LIN {X 0,Y 580.036,Z 777.996,A -85,B 0,C 180,E1 -1980,E2 -1980} C_VEL
LIN {X 0,Y 580.038,Z 777.751,A -85,B 0,C 180,E1 -1980.694,E2 -1980.694} C_VEL
LIN {X 0,Y 580.046,Z 776.958,A -85,B 0,C 180,E1 -1981.389,E2 -1981.389} C_VEL
LIN {X 0,Y 580.034,Z 775.61,A -85,B 0,C 180,E1 -1982.083,E2 -1982.083} C_VEL
LIN {X 0,Y 580.073,Z 772.575,A -85,B 0,C 180,E1 -1983.125,E2 -1983.125} C_VEL
LIN {X 0,Y 580.109,Z 768.035,A -85,B 0,C 180,E1 -1984.169,E2 -1984.169} C_VEL
LIN {X 0,Y 580.127,Z 762.947,A -85,B 0,C 180,E1 -1985.039,E2 -1985.039} C_VEL
LIN {X 0,Y 580.195,Z 756.461,A -85,B 0,C 180,E1 -1985.91,E2 -1985.91} C_VEL
LIN {X 0,Y 580.226,Z 747.843,A -85,B 0,C 180,E1 -1986.806,E2 -1986.806} C_VEL
LIN {X 0,Y 580.271,Z 739.422,A -85,B 0,C 180,E1 -1987.481,E2 -1987.481} C_VEL
LIN {X 0,Y 580.361,Z 729.698,A -85,B 0,C 180,E1 -1988.093,E2 -1988.093} C_VEL
LIN {X 0,Y 580.434,Z 719.272,A -85,B 0,C 180,E1 -1988.574,E2 -1988.574} C_VEL
LIN {X 0,Y 580.421,Z 709.143,A -85,B 0,C 180,E1 -1988.903,E2 -1988.903} C_VEL
LIN {X 0,Y 580.451,Z 698.454,A -85,B 0,C 180,E1 -1989.122,E2 -1989.122} C_VEL
LIN {X 0,Y 580.405,Z 632.513,A -85,B 0,C 180,E1 -1989.936,E2 -1989.936} C_VEL
LIN {X 0,Y 580.269,Z 630.726,A -85,B 0,C 180,E1 -1990.005,E2 -1990.005} C_VEL
LIN {X 0,Y 580.35,Z 617.125,A -85,B 0,C 180,E1 -1991.689,E2 -1991.689} C_VEL
LIN {X 0,Y 579.697,Z 613.548,A -85,B 0,C 180,E1 -1992.149,E2 -1992.149} C_VEL
LIN {X 0,Y 574.108,Z 602.38,A -85,B 0,C 180,E1 -1993.683,E2 -1993.683} C_VEL
LIN {X 0,Y 573.454,Z 598.82,A -85,B 0,C 180,E1 -1994.152,E2 -1994.152} C_VEL
LIN {X 0,Y 573.677,Z 575.438,A -85,B 0,C 180,E1 -1997.144,E2 -1997.144} C_VEL
LIN {X 0,Y 573.912,Z 553.049,A -85,B 0,C 180,E1 -2000.053,E2 -2000.053} C_VEL
LIN {X 0,Y 574.175,Z 533.149,A -85,B 0,C 180,E1 -2002.679,E2 -2002.679} C_VEL
LIN {X 0,Y 574.39,Z 518.935,A -85,B 0,C 180,E1 -2004.583,E2 -2004.583} C_VEL
LIN {X 0,Y 573.29,Z 513.146,A -85,B 0,C 180,E1 -2005.457,E2 -2005.457} C_VEL
LIN {X 0,Y 573.252,Z 513.079,A -85,B 0,C 180,E1 -2008.028,E2 -2008.028} C_VEL
LIN {X 0,Y 573.25,Z 513.08,A -85,B 0,C 180,E1 -2010.176,E2 -2010.176} C_VEL
LIN {X 0,Y 573.258,Z 513.079,A -85,B 0,C 180,E1 -2012.645,E2 -2012.645} C_VEL
LIN {X 0,Y 573.272,Z 513.071,A -85,B 0,C 180,E1 -2015.184,E2 -2015.184} C_VEL
LIN {X 0,Y 573.24,Z 513.075,A -85,B 0,C 180,E1 -2017.807,E2 -2017.807} C_VEL
LIN {X 0,Y 573.275,Z 513.076,A -85,B 0,C 180,E1 -2020.528,E2 -2020.528} C_VEL
LIN {X 0,Y 573.248,Z 513.069,A -85,B 0,C 180,E1 -2023.669,E2 -2023.669} C_VEL
LIN {X 0,Y 573.252,Z 513.081,A -85,B 0,C 180,E1 -2026.642,E2 -2026.642} C_VEL
LIN {X 0,Y 573.249,Z 513.07,A -85,B 0,C 180,E1 -2029.475,E2 -2029.475} C_VEL
LIN {X 0,Y 573.241,Z 513.076,A -85,B 0,C 180,E1 -2032.192,E2 -2032.192} C_VEL
LIN {X 0,Y 573.239,Z 513.074,A -85,B 0,C 180,E1 -2035.229,E2 -2035.229} C_VEL
LIN {X 0,Y 573.257,Z 513.072,A -85,B 0,C 180,E1 -2037.771,E2 -2037.771} C_VEL
LIN {X 0,Y 573.269,Z 513.081,A -85,B 0,C 180,E1 -2040.634,E2 -2040.634} C_VEL
LIN {X 0,Y 573.256,Z 513.077,A -85,B 0,C 180,E1 -2043.024,E2 -2043.024} C_VEL
LIN {X 0,Y 573.281,Z 513.068,A -85,B 0,C 180,E1 -2045.366,E2 -2045.366} C_VEL
LIN {X 0,Y 573.234,Z 513.081,A -85,B 0,C 180,E1 -2048.419,E2 -2048.419} C_VEL
LIN {X 0,Y 573.317,Z 513.261,A -85,B 0,C 180,E1 -2050.276,E2 -2050.276} C_VEL
LIN {X 0,Y 573.558,Z 518.552,A -85,B 0,C 180,E1 -2051.237,E2 -2051.237} C_VEL
LIN {X 0,Y 573.387,Z 536.372,A -85,B 0,C 180,E1 -2054.356,E2 -2054.356} C_VEL
LIN {X 0,Y 573.308,Z 547.196,A -85,B 0,C 180,E1 -2056.192,E2 -2056.192} C_VEL
LIN {X 0,Y 573.776,Z 550.135,A -85,B 0,C 180,E1 -2056.277,E2 -2056.277} C_VEL
LIN {X 0,Y 574.078,Z 556.84,A -85,B 0,C 180,E1 -2056.369,E2 -2056.369} C_VEL
LIN {X 0,Y 573.884,Z 653.913,A -85,B 0,C 180,E1 -2057.602,E2 -2057.602} C_VEL
LIN {X 0,Y 573.815,Z 667.2,A -85,B 0,C 180,E1 -2057.915,E2 -2057.915} C_VEL
LIN {X 0,Y 573.718,Z 679.359,A -85,B 0,C 180,E1 -2058.339,E2 -2058.339} C_VEL
LIN {X 0,Y 573.588,Z 690.955,A -85,B 0,C 180,E1 -2058.881,E2 -2058.881} C_VEL
LIN {X 0,Y 573.447,Z 702.545,A -85,B 0,C 180,E1 -2059.585,E2 -2059.585} C_VEL
LIN {X 0,Y 573.332,Z 713.057,A -85,B 0,C 180,E1 -2060.385,E2 -2060.385} C_VEL
LIN {X 0,Y 573.242,Z 721.659,A -85,B 0,C 180,E1 -2061.184,E2 -2061.184} C_VEL
LIN {X 0,Y 573.162,Z 729.582,A -85,B 0,C 180,E1 -2062.07,E2 -2062.07} C_VEL
LIN {X 0,Y 573.092,Z 737.519,A -85,B 0,C 180,E1 -2063.162,E2 -2063.162} C_VEL
LIN {X 0,Y 573.071,Z 744.446,A -85,B 0,C 180,E1 -2064.369,E2 -2064.369} C_VEL
LIN {X 0,Y 573.028,Z 749.188,A -85,B 0,C 180,E1 -2065.427,E2 -2065.427} C_VEL
LIN {X 0,Y 573.022,Z 752.821,A -85,B 0,C 180,E1 -2066.484,E2 -2066.484} C_VEL
LIN {X 0,Y 572.959,Z 754.699,A -85,B 0,C 180,E1 -2067.187,E2 -2067.187} C_VEL
LIN {X 0,Y 572.939,Z 756.128,A -85,B 0,C 180,E1 -2067.89,E2 -2067.89} C_VEL
LIN {X 0,Y 572.941,Z 757.755,A -85,B 0,C 180,E1 -2069.297,E2 -2069.297} C_VEL
LIN {X 0,Y 572.939,Z 757.996,A -85,B 0,C 180,E1 -2069.999,E2 -2069.999} C_VEL
LIN {X 0,Y 572.94,Z 757.815,A -85,B 0,C 180,E1 -2070.702,E2 -2070.702} C_VEL
LIN {X 0,Y 572.939,Z 756.273,A -85,B 0,C 180,E1 -2072.108,E2 -2072.108} C_VEL
LIN {X 0,Y 572.96,Z 754.912,A -85,B 0,C 180,E1 -2072.812,E2 -2072.812} C_VEL
LIN {X 0,Y 573.015,Z 752.034,A -85,B 0,C 180,E1 -2073.867,E2 -2073.867} C_VEL
LIN {X 0,Y 572.963,Z 748.134,A -85,B 0,C 180,E1 -2074.925,E2 -2074.925} C_VEL
LIN {X 0,Y 573.075,Z 743.102,A -85,B 0,C 180,E1 -2075.983,E2 -2075.983} C_VEL
LIN {X 0,Y 573.082,Z 736.781,A -85,B 0,C 180,E1 -2077.044,E2 -2077.044} C_VEL
LIN {X 0,Y 573.177,Z 728.86,A -85,B 0,C 180,E1 -2078.105,E2 -2078.105} C_VEL
LIN {X 0,Y 573.286,Z 719.011,A -85,B 0,C 180,E1 -2079.17,E2 -2079.17} C_VEL
LIN {X 0,Y 573.424,Z 708.694,A -85,B 0,C 180,E1 -2080.058,E2 -2080.058} C_VEL
LIN {X 0,Y 573.556,Z 697.058,A -85,B 0,C 180,E1 -2080.858,E2 -2080.858} C_VEL
LIN {X 0,Y 573.656,Z 686.213,A -85,B 0,C 180,E1 -2081.449,E2 -2081.449} C_VEL
LIN {X 0,Y 573.754,Z 673.633,A -85,B 0,C 180,E1 -2081.969,E2 -2081.969} C_VEL
LIN {X 0,Y 573.845,Z 660.475,A -85,B 0,C 180,E1 -2082.353,E2 -2082.353} C_VEL
LIN {X 0,Y 573.912,Z 648.143,A -85,B 0,C 180,E1 -2082.576,E2 -2082.576} C_VEL
LIN {X 0,Y 573.908,Z 551.107,A -85,B 0,C 180,E1 -2083.798,E2 -2083.798} C_VEL
LIN {X 0,Y 573.364,Z 547.542,A -85,B 0,C 180,E1 -2083.873,E2 -2083.873} C_VEL
LIN {X 0,Y 573.298,Z 546.336,A -85,B 0,C 180,E1 -2084.011,E2 -2084.011} C_VEL
LIN {X 0,Y 573.451,Z 530.701,A -85,B 0,C 180,E1 -2086.721,E2 -2086.721} C_VEL
LIN {X 0,Y 573.578,Z 515.71,A -85,B 0,C 180,E1 -2089.356,E2 -2089.356} C_VEL
LIN {X 0,Y 573.272,Z 513.185,A -85,B 0,C 180,E1 -2089.841,E2 -2089.841} C_VEL
LIN {X 0,Y 573.238,Z 513.076,A -85,B 0,C 180,E1 -2092.337,E2 -2092.337} C_VEL
LIN {X 0,Y 573.256,Z 513.081,A -85,B 0,C 180,E1 -2095.409,E2 -2095.409} C_VEL
LIN {X 0,Y 573.253,Z 513.074,A -85,B 0,C 180,E1 -2098.028,E2 -2098.028} C_VEL
LIN {X 0,Y 573.239,Z 513.076,A -85,B 0,C 180,E1 -2100.883,E2 -2100.883} C_VEL
LIN {X 0,Y 573.261,Z 513.08,A -85,B 0,C 180,E1 -2103.523,E2 -2103.523} C_VEL
LIN {X 0,Y 573.259,Z 513.072,A -85,B 0,C 180,E1 -2106.047,E2 -2106.047} C_VEL
LIN {X 0,Y 573.247,Z 513.074,A -85,B 0,C 180,E1 -2108.7,E2 -2108.7} C_VEL
LIN {X 0,Y 573.252,Z 513.08,A -85,B 0,C 180,E1 -2111.595,E2 -2111.595} C_VEL
LIN {X 0,Y 573.236,Z 513.073,A -85,B 0,C 180,E1 -2114.332,E2 -2114.332} C_VEL
LIN {X 0,Y 573.236,Z 513.083,A -85,B 0,C 180,E1 -2117.358,E2 -2117.358} C_VEL
LIN {X 0,Y 573.246,Z 513.071,A -85,B 0,C 180,E1 -2120.393,E2 -2120.393} C_VEL
LIN {X 0,Y 573.251,Z 513.075,A -85,B 0,C 180,E1 -2123.077,E2 -2123.077} C_VEL
LIN {X 0,Y 573.27,Z 513.077,A -85,B 0,C 180,E1 -2125.671,E2 -2125.671} C_VEL
LIN {X 0,Y 573.245,Z 513.074,A -85,B 0,C 180,E1 -2128.185,E2 -2128.185} C_VEL
LIN {X 0,Y 573.265,Z 513.071,A -85,B 0,C 180,E1 -2130.634,E2 -2130.634} C_VEL
LIN {X 0,Y 573.265,Z 513.08,A -85,B 0,C 180,E1 -2133.5,E2 -2133.5} C_VEL
LIN {X 0,Y 573.227,Z 513.076,A -85,B 0,C 180,E1 -2136.134,E2 -2136.134} C_VEL
LIN {X 0,Y 573.256,Z 513.076,A -85,B 0,C 180,E1 -2139.174,E2 -2139.174} C_VEL
LIN {X 0,Y 573.233,Z 513.083,A -85,B 0,C 180,E1 -2141.411,E2 -2141.411} C_VEL
LIN {X 0,Y 573.253,Z 513.08,A -85,B 0,C 180,E1 -2143.622,E2 -2143.622} C_VEL
LIN {X 0,Y 573.229,Z 513.075,A -85,B 0,C 180,E1 -2146.529,E2 -2146.529} C_VEL
LIN {X 0,Y 573.255,Z 513.072,A -85,B 0,C 180,E1 -2148.745,E2 -2148.745} C_VEL
LIN {X 0,Y 573.301,Z 513.075,A -85,B 0,C 180,E1 -2151.541,E2 -2151.541} C_VEL
LIN {X 0,Y 573.285,Z 513.068,A -85,B 0,C 180,E1 -2154.372,E2 -2154.372} C_VEL
LIN {X 0,Y 573.303,Z 513.07,A -85,B 0,C 180,E1 -2157.892,E2 -2157.892} C_VEL
LIN {X 0,Y 573.33,Z 513.063,A -85,B 0,C 180,E1 -2160.702,E2 -2160.702} C_VEL
LIN {X 0,Y 573.234,Z 513.083,A -85,B 0,C 180,E1 -2163.514,E2 -2163.514} C_VEL
LIN {X 0,Y 573.284,Z 513.078,A -85,B 0,C 180,E1 -2165.628,E2 -2165.628} C_VEL
LIN {X 0,Y 573.285,Z 513.068,A -85,B 0,C 180,E1 -2168.459,E2 -2168.459} C_VEL
LIN {X 0,Y 573.264,Z 513.075,A -85,B 0,C 180,E1 -2171.312,E2 -2171.312} C_VEL
LIN {X 0,Y 573.266,Z 513.072,A -85,B 0,C 180,E1 -2174.193,E2 -2174.193} C_VEL
LIN {X 0,Y 573.252,Z 513.074,A -85,B 0,C 180,E1 -2177.112,E2 -2177.112} C_VEL
LIN {X 0,Y 573.249,Z 513.075,A -85,B 0,C 180,E1 -2180.077,E2 -2180.077} C_VEL
LIN {X 0,Y 573.231,Z 513.075,A -85,B 0,C 180,E1 -2182.338,E2 -2182.338} C_VEL
LIN {X 0,Y 573.251,Z 513.079,A -85,B 0,C 180,E1 -2185.41,E2 -2185.41} C_VEL
LIN {X 0,Y 573.258,Z 513.076,A -85,B 0,C 180,E1 -2188.032,E2 -2188.032} C_VEL
LIN {X 0,Y 573.232,Z 513.075,A -85,B 0,C 180,E1 -2190.885,E2 -2190.885} C_VEL
LIN {X 0,Y 573.283,Z 513.077,A -85,B 0,C 180,E1 -2193.529,E2 -2193.529} C_VEL
LIN {X 0,Y 573.256,Z 513.073,A -85,B 0,C 180,E1 -2196.049,E2 -2196.049} C_VEL
LIN {X 0,Y 573.244,Z 513.073,A -85,B 0,C 180,E1 -2198.702,E2 -2198.702} C_VEL
LIN {X 0,Y 573.249,Z 513.082,A -85,B 0,C 180,E1 -2201.596,E2 -2201.596} C_VEL
LIN {X 0,Y 573.231,Z 513.076,A -85,B 0,C 180,E1 -2204.334,E2 -2204.334} C_VEL
LIN {X 0,Y 573.248,Z 513.077,A -85,B 0,C 180,E1 -2207.358,E2 -2207.358} C_VEL
LIN {X 0,Y 573.245,Z 513.073,A -85,B 0,C 180,E1 -2210.394,E2 -2210.394} C_VEL
LIN {X 0,Y 573.254,Z 513.071,A -85,B 0,C 180,E1 -2213.079,E2 -2213.079} C_VEL
LIN {X 0,Y 573.266,Z 513.08,A -85,B 0,C 180,E1 -2215.672,E2 -2215.672} C_VEL
LIN {X 0,Y 573.248,Z 513.065,A -85,B 0,C 180,E1 -2218.186,E2 -2218.186} C_VEL
LIN {X 0,Y 573.263,Z 513.071,A -85,B 0,C 180,E1 -2220.635,E2 -2220.635} C_VEL
LIN {X 0,Y 573.251,Z 513.073,A -85,B 0,C 180,E1 -2223.025,E2 -2223.025} C_VEL
LIN {X 0,Y 573.275,Z 513.075,A -85,B 0,C 180,E1 -2225.367,E2 -2225.367} C_VEL
LIN {X 0,Y 573.287,Z 513.31,A -85,B 0,C 180,E1 -2226.936,E2 -2226.936} C_VEL
LIN {X 0,Y 574.008,Z 518.026,A -85,B 0,C 180,E1 -2227.695,E2 -2227.695} C_VEL
LIN {X 0,Y 573.748,Z 538.175,A -85,B 0,C 180,E1 -2230.688,E2 -2230.688} C_VEL
LIN {X 0,Y 573.546,Z 557.107,A -85,B 0,C 180,E1 -2233.454,E2 -2233.454} C_VEL
LIN {X 0,Y 573.395,Z 576.025,A -85,B 0,C 180,E1 -2236.15,E2 -2236.15} C_VEL
LIN {X 0,Y 574.081,Z 581.568,A -85,B 0,C 180,E1 -2236.257,E2 -2236.257} C_VEL
LIN {X 0,Y 573.882,Z 683.983,A -85,B 0,C 180,E1 -2237.558,E2 -2237.558} C_VEL
LIN {X 0,Y 573.811,Z 697.239,A -85,B 0,C 180,E1 -2237.871,E2 -2237.871} C_VEL
LIN {X 0,Y 573.718,Z 709.388,A -85,B 0,C 180,E1 -2238.295,E2 -2238.295} C_VEL
LIN {X 0,Y 573.576,Z 721.729,A -85,B 0,C 180,E1 -2238.879,E2 -2238.879} C_VEL
LIN {X 0,Y 573.438,Z 733.213,A -85,B 0,C 180,E1 -2239.586,E2 -2239.586} C_VEL
LIN {X 0,Y 573.327,Z 743.607,A -85,B 0,C 180,E1 -2240.386,E2 -2240.386} C_VEL
LIN {X 0,Y 573.24,Z 752.12,A -85,B 0,C 180,E1 -2241.185,E2 -2241.185} C_VEL
LIN {X 0,Y 573.16,Z 759.966,A -85,B 0,C 180,E1 -2242.072,E2 -2242.072} C_VEL
LIN {X 0,Y 573.072,Z 767.958,A -85,B 0,C 180,E1 -2243.186,E2 -2243.186} C_VEL
LIN {X 0,Y 573.07,Z 774.683,A -85,B 0,C 180,E1 -2244.37,E2 -2244.37} C_VEL
LIN {X 0,Y 573.028,Z 779.374,A -85,B 0,C 180,E1 -2245.428,E2 -2245.428} C_VEL
LIN {X 0,Y 573.022,Z 782.96,A -85,B 0,C 180,E1 -2246.485,E2 -2246.485} C_VEL
LIN {X 0,Y 572.959,Z 784.811,A -85,B 0,C 180,E1 -2247.188,E2 -2247.188} C_VEL
LIN {X 0,Y 572.937,Z 786.201,A -85,B 0,C 180,E1 -2247.892,E2 -2247.892} C_VEL
LIN {X 0,Y 572.94,Z 787.785,A -85,B 0,C 180,E1 -2249.298,E2 -2249.298} C_VEL
LIN {X 0,Y 572.938,Z 788,A -85,B 0,C 180,E1 -2250.001,E2 -2250.001} C_VEL
LIN {X 0,Y 572.946,Z 787.185,A -85,B 0,C 180,E1 -2251.406,E2 -2251.406} C_VEL
LIN {X 0,Y 572.937,Z 786.198,A -85,B 0,C 180,E1 -2252.11,E2 -2252.11} C_VEL
LIN {X 0,Y 572.959,Z 784.807,A -85,B 0,C 180,E1 -2252.813,E2 -2252.813} C_VEL
LIN {X 0,Y 573.014,Z 781.893,A -85,B 0,C 180,E1 -2253.869,E2 -2253.869} C_VEL
LIN {X 0,Y 572.963,Z 777.947,A -85,B 0,C 180,E1 -2254.926,E2 -2254.926} C_VEL
LIN {X 0,Y 573.064,Z 771.873,A -85,B 0,C 180,E1 -2256.161,E2 -2256.161} C_VEL
LIN {X 0,Y 573.12,Z 765.233,A -85,B 0,C 180,E1 -2257.221,E2 -2257.221} C_VEL
LIN {X 0,Y 573.201,Z 756.986,A -85,B 0,C 180,E1 -2258.284,E2 -2258.284} C_VEL
LIN {X 0,Y 573.287,Z 748.532,A -85,B 0,C 180,E1 -2259.171,E2 -2259.171} C_VEL
LIN {X 0,Y 573.409,Z 738.09,A -85,B 0,C 180,E1 -2260.059,E2 -2260.059} C_VEL
LIN {X 0,Y 573.55,Z 726.343,A -85,B 0,C 180,E1 -2260.858,E2 -2260.858} C_VEL
LIN {X 0,Y 573.654,Z 715.27,A -85,B 0,C 180,E1 -2261.448,E2 -2261.448} C_VEL
LIN {X 0,Y 573.767,Z 702.162,A -85,B 0,C 180,E1 -2261.974,E2 -2261.974} C_VEL
LIN {X 0,Y 573.836,Z 689.5,A -85,B 0,C 180,E1 -2262.332,E2 -2262.332} C_VEL
LIN {X 0,Y 573.932,Z 676.265,A -85,B 0,C 180,E1 -2262.554,E2 -2262.554} C_VEL
LIN {X 0,Y 573.931,Z 579.676,A -85,B 0,C 180,E1 -2263.77,E2 -2263.77} C_VEL
LIN {X 0,Y 573.407,Z 576.004,A -85,B 0,C 180,E1 -2263.851,E2 -2263.851} C_VEL
LIN {X 0,Y 573.548,Z 555.883,A -85,B 0,C 180,E1 -2266.724,E2 -2266.724} C_VEL
LIN {X 0,Y 573.741,Z 537.567,A -85,B 0,C 180,E1 -2269.402,E2 -2269.402} C_VEL
LIN {X 0,Y 574.002,Z 518.017,A -85,B 0,C 180,E1 -2272.307,E2 -2272.307} C_VEL
LIN {X 0,Y 573.242,Z 513.207,A -85,B 0,C 180,E1 -2273.1,E2 -2273.1} C_VEL
LIN {X 0,Y 573.253,Z 513.074,A -85,B 0,C 180,E1 -2275.411,E2 -2275.411} C_VEL
LIN {X 0,Y 573.255,Z 513.081,A -85,B 0,C 180,E1 -2278.029,E2 -2278.029} C_VEL
LIN {X 0,Y 573.25,Z 513.08,A -85,B 0,C 180,E1 -2280.176,E2 -2280.176} C_VEL
LIN {X 0,Y 573.257,Z 513.075,A -85,B 0,C 180,E1 -2282.645,E2 -2282.645} C_VEL
LIN {X 0,Y 573.21,Z 513.078,A -85,B 0,C 180,E1 -2285.188,E2 -2285.188} C_VEL
LIN {X 0,Y 573.24,Z 513.08,A -85,B 0,C 180,E1 -2287.808,E2 -2287.808} C_VEL
LIN {X 0,Y 573.249,Z 513.076,A -85,B 0,C 180,E1 -2290.525,E2 -2290.525} C_VEL
LIN {X 0,Y 573.257,Z 513.077,A -85,B 0,C 180,E1 -2293.67,E2 -2293.67} C_VEL
LIN {X 0,Y 573.243,Z 513.075,A -85,B 0,C 180,E1 -2296.641,E2 -2296.641} C_VEL
LIN {X 0,Y 573.263,Z 513.075,A -85,B 0,C 180,E1 -2299.476,E2 -2299.476} C_VEL
LIN {X 0,Y 573.24,Z 513.08,A -85,B 0,C 180,E1 -2302.193,E2 -2302.193} C_VEL
LIN {X 0,Y 573.272,Z 513.071,A -85,B 0,C 180,E1 -2304.817,E2 -2304.817} C_VEL
LIN {X 0,Y 573.258,Z 513.076,A -85,B 0,C 180,E1 -2307.355,E2 -2307.355} C_VEL
LIN {X 0,Y 573.251,Z 513.075,A -85,B 0,C 180,E1 -2310.512,E2 -2310.512} C_VEL
LIN {X 0,Y 573.252,Z 513.076,A -85,B 0,C 180,E1 -2313.024,E2 -2313.024} C_VEL
LIN {X 0,Y 573.297,Z 513.239,A -85,B 0,C 180,E1 -2314.659,E2 -2314.659} C_VEL
LIN {X 0,Y 574.313,Z 518.272,A -85,B 0,C 180,E1 -2315.414,E2 -2315.414} C_VEL
LIN {X 0,Y 574.212,Z 531.056,A -85,B 0,C 180,E1 -2317.132,E2 -2317.132} C_VEL
LIN {X 0,Y 573.919,Z 552.364,A -85,B 0,C 180,E1 -2319.948,E2 -2319.948} C_VEL
LIN {X 0,Y 573.698,Z 573.817,A -85,B 0,C 180,E1 -2322.737,E2 -2322.737} C_VEL
LIN {X 0,Y 573.445,Z 596.558,A -85,B 0,C 180,E1 -2325.65,E2 -2325.65} C_VEL
LIN {X 0,Y 573.322,Z 619.136,A -85,B 0,C 180,E1 -2328.51,E2 -2328.51} C_VEL
LIN {X 0,Y 573.24,Z 630.977,A -85,B 0,C 180,E1 -2329.983,E2 -2329.983} C_VEL
LIN {X 0,Y 573.561,Z 635.98,A -85,B 0,C 180,E1 -2330.078,E2 -2330.078} C_VEL
LIN {X 0,Y 573.479,Z 702.327,A -85,B 0,C 180,E1 -2330.922,E2 -2330.922} C_VEL
LIN {X 0,Y 573.425,Z 714.415,A -85,B 0,C 180,E1 -2331.232,E2 -2331.232} C_VEL
LIN {X 0,Y 573.351,Z 724.357,A -85,B 0,C 180,E1 -2331.63,E2 -2331.63} C_VEL
LIN {X 0,Y 573.286,Z 734.166,A -85,B 0,C 180,E1 -2332.161,E2 -2332.161} C_VEL
LIN {X 0,Y 573.195,Z 744.026,A -85,B 0,C 180,E1 -2332.869,E2 -2332.869} C_VEL
LIN {X 0,Y 573.14,Z 751.59,A -85,B 0,C 180,E1 -2333.568,E2 -2333.568} C_VEL
LIN {X 0,Y 573.087,Z 758.58,A -85,B 0,C 180,E1 -2334.37,E2 -2334.37} C_VEL
LIN {X 0,Y 573.081,Z 765.654,A -85,B 0,C 180,E1 -2335.428,E2 -2335.428} C_VEL
LIN {X 0,Y 573.055,Z 770.835,A -85,B 0,C 180,E1 -2336.484,E2 -2336.484} C_VEL
LIN {X 0,Y 572.971,Z 773.435,A -85,B 0,C 180,E1 -2337.188,E2 -2337.188} C_VEL
LIN {X 0,Y 572.936,Z 775.407,A -85,B 0,C 180,E1 -2337.891,E2 -2337.891} C_VEL
LIN {X 0,Y 572.942,Z 776.834,A -85,B 0,C 180,E1 -2338.594,E2 -2338.594} C_VEL
LIN {X 0,Y 572.936,Z 777.691,A -85,B 0,C 180,E1 -2339.297,E2 -2339.297} C_VEL
LIN {X 0,Y 572.936,Z 777.996,A -85,B 0,C 180,E1 -2340,E2 -2340} C_VEL
LIN {X 0,Y 572.938,Z 777.754,A -85,B 0,C 180,E1 -2340.703,E2 -2340.703} C_VEL
LIN {X 0,Y 572.946,Z 776.962,A -85,B 0,C 180,E1 -2341.406,E2 -2341.406} C_VEL
LIN {X 0,Y 572.935,Z 775.612,A -85,B 0,C 180,E1 -2342.109,E2 -2342.109} C_VEL
LIN {X 0,Y 572.993,Z 772.574,A -85,B 0,C 180,E1 -2343.164,E2 -2343.164} C_VEL
LIN {X 0,Y 573.039,Z 768.032,A -85,B 0,C 180,E1 -2344.22,E2 -2344.22} C_VEL
LIN {X 0,Y 573.027,Z 762.949,A -85,B 0,C 180,E1 -2345.101,E2 -2345.101} C_VEL
LIN {X 0,Y 573.139,Z 756.463,A -85,B 0,C 180,E1 -2345.983,E2 -2345.983} C_VEL
LIN {X 0,Y 573.163,Z 748.225,A -85,B 0,C 180,E1 -2346.855,E2 -2346.855} C_VEL
LIN {X 0,Y 573.236,Z 739.423,A -85,B 0,C 180,E1 -2347.574,E2 -2347.574} C_VEL
LIN {X 0,Y 573.337,Z 729.691,A -85,B 0,C 180,E1 -2348.193,E2 -2348.193} C_VEL
LIN {X 0,Y 573.396,Z 719.261,A -85,B 0,C 180,E1 -2348.68,E2 -2348.68} C_VEL
LIN {X 0,Y 573.42,Z 709.141,A -85,B 0,C 180,E1 -2349.013,E2 -2349.013} C_VEL
LIN {X 0,Y 573.455,Z 698.416,A -85,B 0,C 180,E1 -2349.234,E2 -2349.234} C_VEL
LIN {X 0,Y 573.452,Z 633.363,A -85,B 0,C 180,E1 -2350.047,E2 -2350.047} C_VEL
LIN {X 0,Y 573.25,Z 630.983,A -85,B 0,C 180,E1 -2350.106,E2 -2350.106} C_VEL
LIN {X 0,Y 573.4,Z 607.058,A -85,B 0,C 180,E1 -2353.106,E2 -2353.106} C_VEL
LIN {X 0,Y 573.454,Z 598.82,A -85,B 0,C 180,E1 -2354.152,E2 -2354.152} C_VEL
LIN {X 0,Y 572.787,Z 595.28,A -85,B 0,C 180,E1 -2354.62,E2 -2354.62} C_VEL
LIN {X 0,Y 567.216,Z 584.309,A -85,B 0,C 180,E1 -2356.188,E2 -2356.188} C_VEL
LIN {X 0,Y 566.655,Z 580.776,A -85,B 0,C 180,E1 -2356.665,E2 -2356.665} C_VEL
LIN {X 0,Y 566.955,Z 558.442,A -85,B 0,C 180,E1 -2359.592,E2 -2359.592} C_VEL
LIN {X 0,Y 567.273,Z 535.987,A -85,B 0,C 180,E1 -2362.586,E2 -2362.586} C_VEL
LIN {X 0,Y 567.457,Z 520.098,A -85,B 0,C 180,E1 -2364.708,E2 -2364.708} C_VEL
LIN {X 0,Y 566.226,Z 514.034,A -85,B 0,C 180,E1 -2365.578,E2 -2365.578} C_VEL
LIN {X 0,Y 566.207,Z 513.959,A -85,B 0,C 180,E1 -2368.202,E2 -2368.202} C_VEL
LIN {X 0,Y 566.194,Z 513.954,A -85,B 0,C 180,E1 -2371.076,E2 -2371.076} C_VEL
LIN {X 0,Y 566.217,Z 513.95,A -85,B 0,C 180,E1 -2373.734,E2 -2373.734} C_VEL
LIN {X 0,Y 566.221,Z 513.957,A -85,B 0,C 180,E1 -2376.569,E2 -2376.569} C_VEL
LIN {X 0,Y 566.216,Z 513.949,A -85,B 0,C 180,E1 -2379.685,E2 -2379.685} C_VEL
LIN {X 0,Y 566.193,Z 513.952,A -85,B 0,C 180,E1 -2382.09,E2 -2382.09} C_VEL
LIN {X 0,Y 566.179,Z 513.955,A -85,B 0,C 180,E1 -2385.036,E2 -2385.036} C_VEL
LIN {X 0,Y 566.224,Z 513.952,A -85,B 0,C 180,E1 -2388.136,E2 -2388.136} C_VEL
LIN {X 0,Y 566.224,Z 513.954,A -85,B 0,C 180,E1 -2390.727,E2 -2390.727} C_VEL
LIN {X 0,Y 566.189,Z 513.953,A -85,B 0,C 180,E1 -2393.788,E2 -2393.788} C_VEL
LIN {X 0,Y 566.217,Z 513.952,A -85,B 0,C 180,E1 -2396.266,E2 -2396.266} C_VEL
LIN {X 0,Y 566.198,Z 513.957,A -85,B 0,C 180,E1 -2398.923,E2 -2398.923} C_VEL
LIN {X 0,Y 566.217,Z 513.949,A -85,B 0,C 180,E1 -2401.857,E2 -2401.857} C_VEL
LIN {X 0,Y 566.218,Z 513.953,A -85,B 0,C 180,E1 -2404.251,E2 -2404.251} C_VEL
LIN {X 0,Y 566.196,Z 513.961,A -85,B 0,C 180,E1 -2406.714,E2 -2406.714} C_VEL
LIN {X 0,Y 566.222,Z 513.956,A -85,B 0,C 180,E1 -2409.663,E2 -2409.663} C_VEL
LIN {X 0,Y 566.288,Z 514.172,A -85,B 0,C 180,E1 -2410.186,E2 -2410.186} C_VEL
LIN {X 0,Y 566.542,Z 520.652,A -85,B 0,C 180,E1 -2411.371,E2 -2411.371} C_VEL
LIN {X 0,Y 566.352,Z 537.423,A -85,B 0,C 180,E1 -2414.341,E2 -2414.341} C_VEL
LIN {X 0,Y 566.278,Z 547.213,A -85,B 0,C 180,E1 -2416.017,E2 -2416.017} C_VEL
LIN {X 0,Y 566.867,Z 550.851,A -85,B 0,C 180,E1 -2416.115,E2 -2416.115} C_VEL
LIN {X 0,Y 567.18,Z 556.885,A -85,B 0,C 180,E1 -2416.2,E2 -2416.2} C_VEL
LIN {X 0,Y 566.964,Z 653.942,A -85,B 0,C 180,E1 -2417.448,E2 -2417.448} C_VEL
LIN {X 0,Y 566.877,Z 667.219,A -85,B 0,C 180,E1 -2417.764,E2 -2417.764} C_VEL
LIN {X 0,Y 566.751,Z 679.375,A -85,B 0,C 180,E1 -2418.193,E2 -2418.193} C_VEL
LIN {X 0,Y 566.606,Z 691.636,A -85,B 0,C 180,E1 -2418.78,E2 -2418.78} C_VEL
LIN {X 0,Y 566.438,Z 703.841,A -85,B 0,C 180,E1 -2419.545,E2 -2419.545} C_VEL
LIN {X 0,Y 566.299,Z 714.125,A -85,B 0,C 180,E1 -2420.355,E2 -2420.355} C_VEL
LIN {X 0,Y 566.183,Z 723.374,A -85,B 0,C 180,E1 -2421.253,E2 -2421.253} C_VEL
LIN {X 0,Y 566.082,Z 732.345,A -85,B 0,C 180,E1 -2422.33,E2 -2422.33} C_VEL
LIN {X 0,Y 566.01,Z 739.456,A -85,B 0,C 180,E1 -2423.386,E2 -2423.386} C_VEL
LIN {X 0,Y 566.004,Z 744.449,A -85,B 0,C 180,E1 -2424.299,E2 -2424.299} C_VEL
LIN {X 0,Y 565.933,Z 749.191,A -85,B 0,C 180,E1 -2425.369,E2 -2425.369} C_VEL
LIN {X 0,Y 565.927,Z 752.824,A -85,B 0,C 180,E1 -2426.439,E2 -2426.439} C_VEL
LIN {X 0,Y 565.878,Z 754.701,A -85,B 0,C 180,E1 -2427.152,E2 -2427.152} C_VEL
LIN {X 0,Y 565.84,Z 756.128,A -85,B 0,C 180,E1 -2427.864,E2 -2427.864} C_VEL
LIN {X 0,Y 565.841,Z 757.755,A -85,B 0,C 180,E1 -2429.288,E2 -2429.288} C_VEL
LIN {X 0,Y 565.839,Z 757.996,A -85,B 0,C 180,E1 -2429.999,E2 -2429.999} C_VEL
LIN {X 0,Y 565.841,Z 757.815,A -85,B 0,C 180,E1 -2430.711,E2 -2430.711} C_VEL
LIN {X 0,Y 565.84,Z 756.272,A -85,B 0,C 180,E1 -2432.135,E2 -2432.135} C_VEL
LIN {X 0,Y 565.878,Z 754.911,A -85,B 0,C 180,E1 -2432.847,E2 -2432.847} C_VEL
LIN {X 0,Y 565.927,Z 752.032,A -85,B 0,C 180,E1 -2433.916,E2 -2433.916} C_VEL
LIN {X 0,Y 565.878,Z 748.132,A -85,B 0,C 180,E1 -2434.987,E2 -2434.987} C_VEL
LIN {X 0,Y 565.99,Z 743.1,A -85,B 0,C 180,E1 -2436.058,E2 -2436.058} C_VEL
LIN {X 0,Y 566.03,Z 736.777,A -85,B 0,C 180,E1 -2437.132,E2 -2437.132} C_VEL
LIN {X 0,Y 566.132,Z 728.855,A -85,B 0,C 180,E1 -2438.207,E2 -2438.207} C_VEL
LIN {X 0,Y 566.249,Z 719.005,A -85,B 0,C 180,E1 -2439.285,E2 -2439.285} C_VEL
LIN {X 0,Y 566.424,Z 708.688,A -85,B 0,C 180,E1 -2440.183,E2 -2440.183} C_VEL
LIN {X 0,Y 566.562,Z 697.411,A -85,B 0,C 180,E1 -2440.971,E2 -2440.971} C_VEL
LIN {X 0,Y 566.687,Z 686.201,A -85,B 0,C 180,E1 -2441.591,E2 -2441.591} C_VEL
LIN {X 0,Y 566.816,Z 673.618,A -85,B 0,C 180,E1 -2442.118,E2 -2442.118} C_VEL
LIN {X 0,Y 566.935,Z 660.452,A -85,B 0,C 180,E1 -2442.506,E2 -2442.506} C_VEL
LIN {X 0,Y 567.004,Z 648.102,A -85,B 0,C 180,E1 -2442.732,E2 -2442.732} C_VEL
LIN {X 0,Y 567.091,Z 552.305,A -85,B 0,C 180,E1 -2443.951,E2 -2443.951} C_VEL
LIN {X 0,Y 566.306,Z 547.546,A -85,B 0,C 180,E1 -2444.05,E2 -2444.05} C_VEL
LIN {X 0,Y 566.272,Z 546.336,A -85,B 0,C 180,E1 -2444.188,E2 -2444.188} C_VEL
LIN {X 0,Y 566.442,Z 529.292,A -85,B 0,C 180,E1 -2447.183,E2 -2447.183} C_VEL
LIN {X 0,Y 566.526,Z 515.919,A -85,B 0,C 180,E1 -2449.568,E2 -2449.568} C_VEL
LIN {X 0,Y 566.236,Z 514.029,A -85,B 0,C 180,E1 -2449.957,E2 -2449.957} C_VEL
LIN {X 0,Y 566.18,Z 513.956,A -85,B 0,C 180,E1 -2452.631,E2 -2452.631} C_VEL
LIN {X 0,Y 566.218,Z 513.954,A -85,B 0,C 180,E1 -2455.029,E2 -2455.029} C_VEL
LIN {X 0,Y 566.212,Z 513.958,A -85,B 0,C 180,E1 -2457.338,E2 -2457.338} C_VEL
LIN {X 0,Y 566.202,Z 513.954,A -85,B 0,C 180,E1 -2459.768,E2 -2459.768} C_VEL
LIN {X 0,Y 566.206,Z 513.95,A -85,B 0,C 180,E1 -2462.43,E2 -2462.43} C_VEL
LIN {X 0,Y 566.21,Z 513.954,A -85,B 0,C 180,E1 -2464.993,E2 -2464.993} C_VEL
LIN {X 0,Y 566.195,Z 513.961,A -85,B 0,C 180,E1 -2467.46,E2 -2467.46} C_VEL
LIN {X 0,Y 566.225,Z 513.947,A -85,B 0,C 180,E1 -2470.196,E2 -2470.196} C_VEL
LIN {X 0,Y 566.203,Z 513.955,A -85,B 0,C 180,E1 -2473.053,E2 -2473.053} C_VEL
LIN {X 0,Y 566.194,Z 513.953,A -85,B 0,C 180,E1 -2476.048,E2 -2476.048} C_VEL
LIN {X 0,Y 566.208,Z 513.952,A -85,B 0,C 180,E1 -2478.863,E2 -2478.863} C_VEL
LIN {X 0,Y 566.186,Z 513.958,A -85,B 0,C 180,E1 -2481.637,E2 -2481.637} C_VEL
LIN {X 0,Y 566.208,Z 513.95,A -85,B 0,C 180,E1 -2484.311,E2 -2484.311} C_VEL
LIN {X 0,Y 566.224,Z 513.95,A -85,B 0,C 180,E1 -2486.898,E2 -2486.898} C_VEL
LIN {X 0,Y 566.189,Z 513.961,A -85,B 0,C 180,E1 -2489.408,E2 -2489.408} C_VEL
LIN {X 0,Y 566.222,Z 513.951,A -85,B 0,C 180,E1 -2491.858,E2 -2491.858} C_VEL
LIN {X 0,Y 566.221,Z 513.949,A -85,B 0,C 180,E1 -2494.251,E2 -2494.251} C_VEL
LIN {X 0,Y 566.185,Z 513.953,A -85,B 0,C 180,E1 -2496.713,E2 -2496.713} C_VEL
LIN {X 0,Y 566.214,Z 513.956,A -85,B 0,C 180,E1 -2499.663,E2 -2499.663} C_VEL
LIN {X 0,Y 566.198,Z 513.95,A -85,B 0,C 180,E1 -2502.668,E2 -2502.668} C_VEL
LIN {X 0,Y 566.227,Z 513.956,A -85,B 0,C 180,E1 -2505.627,E2 -2505.627} C_VEL
LIN {X 0,Y 566.227,Z 513.947,A -85,B 0,C 180,E1 -2508.675,E2 -2508.675} C_VEL
LIN {X 0,Y 566.241,Z 513.952,A -85,B 0,C 180,E1 -2511.434,E2 -2511.434} C_VEL
LIN {X 0,Y 566.253,Z 513.945,A -85,B 0,C 180,E1 -2514.302,E2 -2514.302} C_VEL
LIN {X 0,Y 566.274,Z 513.946,A -85,B 0,C 180,E1 -2517.866,E2 -2517.866} C_VEL
LIN {X 0,Y 566.3,Z 513.939,A -85,B 0,C 180,E1 -2520.711,E2 -2520.711} C_VEL
LIN {X 0,Y 566.272,Z 513.941,A -85,B 0,C 180,E1 -2522.846,E2 -2522.846} C_VEL
LIN {X 0,Y 566.252,Z 513.952,A -85,B 0,C 180,E1 -2525.698,E2 -2525.698} C_VEL
LIN {X 0,Y 566.228,Z 513.947,A -85,B 0,C 180,E1 -2528.566,E2 -2528.566} C_VEL
LIN {X 0,Y 566.234,Z 513.953,A -85,B 0,C 180,E1 -2531.454,E2 -2531.454} C_VEL
LIN {X 0,Y 566.227,Z 513.947,A -85,B 0,C 180,E1 -2534.507,E2 -2534.507} C_VEL
LIN {X 0,Y 566.197,Z 513.955,A -85,B 0,C 180,E1 -2537.332,E2 -2537.332} C_VEL
LIN {X 0,Y 566.212,Z 513.949,A -85,B 0,C 180,E1 -2540.337,E2 -2540.337} C_VEL
LIN {X 0,Y 566.182,Z 513.959,A -85,B 0,C 180,E1 -2543.404,E2 -2543.404} C_VEL
LIN {X 0,Y 566.22,Z 513.955,A -85,B 0,C 180,E1 -2545.749,E2 -2545.749} C_VEL
LIN {X 0,Y 566.2,Z 513.953,A -85,B 0,C 180,E1 -2548.204,E2 -2548.204} C_VEL
LIN {X 0,Y 566.193,Z 513.953,A -85,B 0,C 180,E1 -2551.079,E2 -2551.079} C_VEL
LIN {X 0,Y 566.217,Z 513.953,A -85,B 0,C 180,E1 -2553.956,E2 -2553.956} C_VEL
LIN {X 0,Y 566.211,Z 513.946,A -85,B 0,C 180,E1 -2556.569,E2 -2556.569} C_VEL
LIN {X 0,Y 566.208,Z 513.96,A -85,B 0,C 180,E1 -2559.686,E2 -2559.686} C_VEL
LIN {X 0,Y 566.209,Z 513.951,A -85,B 0,C 180,E1 -2562.088,E2 -2562.088} C_VEL
LIN {X 0,Y 566.169,Z 513.956,A -85,B 0,C 180,E1 -2565.037,E2 -2565.037} C_VEL
LIN {X 0,Y 566.214,Z 513.956,A -85,B 0,C 180,E1 -2567.914,E2 -2567.914} C_VEL
LIN {X 0,Y 566.219,Z 513.947,A -85,B 0,C 180,E1 -2570.728,E2 -2570.728} C_VEL
LIN {X 0,Y 566.204,Z 513.96,A -85,B 0,C 180,E1 -2573.786,E2 -2573.786} C_VEL
LIN {X 0,Y 566.228,Z 513.946,A -85,B 0,C 180,E1 -2576.899,E2 -2576.899} C_VEL
LIN {X 0,Y 566.186,Z 513.945,A -85,B 0,C 180,E1 -2579.409,E2 -2579.409} C_VEL
LIN {X 0,Y 566.228,Z 513.955,A -85,B 0,C 180,E1 -2581.859,E2 -2581.859} C_VEL
LIN {X 0,Y 566.213,Z 513.95,A -85,B 0,C 180,E1 -2584.252,E2 -2584.252} C_VEL
LIN {X 0,Y 566.212,Z 514.098,A -85,B 0,C 180,E1 -2586.741,E2 -2586.741} C_VEL
LIN {X 0,Y 567.096,Z 519.286,A -85,B 0,C 180,E1 -2587.6,E2 -2587.6} C_VEL
LIN {X 0,Y 566.788,Z 539.048,A -85,B 0,C 180,E1 -2590.571,E2 -2590.571} C_VEL
LIN {X 0,Y 566.562,Z 557.208,A -85,B 0,C 180,E1 -2593.259,E2 -2593.259} C_VEL
LIN {X 0,Y 566.406,Z 576.031,A -85,B 0,C 180,E1 -2595.976,E2 -2595.976} C_VEL
LIN {X 0,Y 567.208,Z 582.361,A -85,B 0,C 180,E1 -2596.098,E2 -2596.098} C_VEL
LIN {X 0,Y 566.972,Z 683.983,A -85,B 0,C 180,E1 -2597.404,E2 -2597.404} C_VEL
LIN {X 0,Y 566.866,Z 697.237,A -85,B 0,C 180,E1 -2597.72,E2 -2597.72} C_VEL
LIN {X 0,Y 566.762,Z 709.388,A -85,B 0,C 180,E1 -2598.149,E2 -2598.149} C_VEL
LIN {X 0,Y 566.626,Z 721.167,A -85,B 0,C 180,E1 -2598.709,E2 -2598.709} C_VEL
LIN {X 0,Y 566.459,Z 733.212,A -85,B 0,C 180,E1 -2599.456,E2 -2599.456} C_VEL
LIN {X 0,Y 566.319,Z 743.609,A -85,B 0,C 180,E1 -2600.266,E2 -2600.266} C_VEL
LIN {X 0,Y 566.207,Z 752.12,A -85,B 0,C 180,E1 -2601.075,E2 -2601.075} C_VEL
LIN {X 0,Y 566.112,Z 759.966,A -85,B 0,C 180,E1 -2601.972,E2 -2601.972} C_VEL
LIN {X 0,Y 566.003,Z 767.626,A -85,B 0,C 180,E1 -2603.047,E2 -2603.047} C_VEL
LIN {X 0,Y 566.003,Z 774.683,A -85,B 0,C 180,E1 -2604.3,E2 -2604.3} C_VEL
LIN {X 0,Y 565.933,Z 779.374,A -85,B 0,C 180,E1 -2605.371,E2 -2605.371} C_VEL
LIN {X 0,Y 565.927,Z 782.961,A -85,B 0,C 180,E1 -2606.441,E2 -2606.441} C_VEL
LIN {X 0,Y 565.878,Z 784.811,A -85,B 0,C 180,E1 -2607.153,E2 -2607.153} C_VEL
LIN {X 0,Y 565.846,Z 787.187,A -85,B 0,C 180,E1 -2608.577,E2 -2608.577} C_VEL
LIN {X 0,Y 565.839,Z 788,A -85,B 0,C 180,E1 -2610.001,E2 -2610.001} C_VEL
LIN {X 0,Y 565.846,Z 787.185,A -85,B 0,C 180,E1 -2611.424,E2 -2611.424} C_VEL
LIN {X 0,Y 565.878,Z 784.807,A -85,B 0,C 180,E1 -2612.848,E2 -2612.848} C_VEL
LIN {X 0,Y 565.926,Z 781.893,A -85,B 0,C 180,E1 -2613.917,E2 -2613.917} C_VEL
LIN {X 0,Y 565.878,Z 777.947,A -85,B 0,C 180,E1 -2614.988,E2 -2614.988} C_VEL
LIN {X 0,Y 566.002,Z 772.864,A -85,B 0,C 180,E1 -2616.059,E2 -2616.059} C_VEL
LIN {X 0,Y 566.041,Z 766.464,A -85,B 0,C 180,E1 -2617.133,E2 -2617.133} C_VEL
LIN {X 0,Y 566.134,Z 758.473,A -85,B 0,C 180,E1 -2618.208,E2 -2618.208} C_VEL
LIN {X 0,Y 566.229,Z 750.33,A -85,B 0,C 180,E1 -2619.106,E2 -2619.106} C_VEL
LIN {X 0,Y 566.339,Z 740.394,A -85,B 0,C 180,E1 -2620.006,E2 -2620.006} C_VEL
LIN {X 0,Y 566.526,Z 729.279,A -85,B 0,C 180,E1 -2620.808,E2 -2620.808} C_VEL
LIN {X 0,Y 566.614,Z 718.165,A -85,B 0,C 180,E1 -2621.447,E2 -2621.447} C_VEL
LIN {X 0,Y 566.75,Z 705.975,A -85,B 0,C 180,E1 -2621.988,E2 -2621.988} C_VEL
LIN {X 0,Y 566.916,Z 693.159,A -85,B 0,C 180,E1 -2622.394,E2 -2622.394} C_VEL
LIN {X 0,Y 566.992,Z 679.564,A -85,B 0,C 180,E1 -2622.665,E2 -2622.665} C_VEL
LIN {X 0,Y 567.033,Z 580.378,A -85,B 0,C 180,E1 -2623.932,E2 -2623.932} C_VEL
LIN {X 0,Y 566.399,Z 576.01,A -85,B 0,C 180,E1 -2624.026,E2 -2624.026} C_VEL
LIN {X 0,Y 566.573,Z 556.082,A -85,B 0,C 180,E1 -2626.906,E2 -2626.906} C_VEL
LIN {X 0,Y 566.83,Z 536.907,A -85,B 0,C 180,E1 -2629.747,E2 -2629.747} C_VEL
LIN {X 0,Y 567.078,Z 519.276,A -85,B 0,C 180,E1 -2632.402,E2 -2632.402} C_VEL
LIN {X 0,Y 566.189,Z 514.054,A -85,B 0,C 180,E1 -2633.285,E2 -2633.285} C_VEL
LIN {X 0,Y 566.214,Z 513.952,A -85,B 0,C 180,E1 -2635.749,E2 -2635.749} C_VEL
LIN {X 0,Y 566.207,Z 513.954,A -85,B 0,C 180,E1 -2638.202,E2 -2638.202} C_VEL
LIN {X 0,Y 566.195,Z 513.953,A -85,B 0,C 180,E1 -2641.077,E2 -2641.077} C_VEL
LIN {X 0,Y 566.216,Z 513.954,A -85,B 0,C 180,E1 -2643.734,E2 -2643.734} C_VEL
LIN {X 0,Y 566.203,Z 513.953,A -85,B 0,C 180,E1 -2646.57,E2 -2646.57} C_VEL
LIN {X 0,Y 566.22,Z 513.953,A -85,B 0,C 180,E1 -2649.686,E2 -2649.686} C_VEL
LIN {X 0,Y 566.219,Z 513.958,A -85,B 0,C 180,E1 -2652.087,E2 -2652.087} C_VEL
LIN {X 0,Y 566.178,Z 513.954,A -85,B 0,C 180,E1 -2655.036,E2 -2655.036} C_VEL
LIN {X 0,Y 566.222,Z 513.956,A -85,B 0,C 180,E1 -2658.136,E2 -2658.136} C_VEL
LIN {X 0,Y 566.225,Z 513.948,A -85,B 0,C 180,E1 -2660.727,E2 -2660.727} C_VEL
LIN {X 0,Y 566.222,Z 513.958,A -85,B 0,C 180,E1 -2663.784,E2 -2663.784} C_VEL
LIN {X 0,Y 566.216,Z 513.953,A -85,B 0,C 180,E1 -2666.266,E2 -2666.266} C_VEL
LIN {X 0,Y 566.194,Z 513.953,A -85,B 0,C 180,E1 -2668.924,E2 -2668.924} C_VEL
LIN {X 0,Y 566.215,Z 513.959,A -85,B 0,C 180,E1 -2671.857,E2 -2671.857} C_VEL
LIN {X 0,Y 566.255,Z 514.138,A -85,B 0,C 180,E1 -2674.605,E2 -2674.605} C_VEL
LIN {X 0,Y 567.453,Z 520.737,A -85,B 0,C 180,E1 -2675.487,E2 -2675.487} C_VEL
LIN {X 0,Y 567.296,Z 533.902,A -85,B 0,C 180,E1 -2677.223,E2 -2677.223} C_VEL
LIN {X 0,Y 566.979,Z 555.213,A -85,B 0,C 180,E1 -2680.07,E2 -2680.07} C_VEL
LIN {X 0,Y 566.719,Z 576.416,A -85,B 0,C 180,E1 -2682.857,E2 -2682.857} C_VEL
LIN {X 0,Y 566.458,Z 600.671,A -85,B 0,C 180,E1 -2685.999,E2 -2685.999} C_VEL
LIN {X 0,Y 566.283,Z 626.244,A -85,B 0,C 180,E1 -2689.271,E2 -2689.271} C_VEL
LIN {X 0,Y 566.208,Z 630.99,A -85,B 0,C 180,E1 -2689.857,E2 -2689.857} C_VEL
LIN {X 0,Y 566.568,Z 636.025,A -85,B 0,C 180,E1 -2689.954,E2 -2689.954} C_VEL
LIN {X 0,Y 566.468,Z 702.388,A -85,B 0,C 180,E1 -2690.808,E2 -2690.808} C_VEL
LIN {X 0,Y 566.426,Z 714.431,A -85,B 0,C 180,E1 -2691.123,E2 -2691.123} C_VEL
LIN {X 0,Y 566.346,Z 724.382,A -85,B 0,C 180,E1 -2691.526,E2 -2691.526} C_VEL
LIN {X 0,Y 566.243,Z 734.184,A -85,B 0,C 180,E1 -2692.063,E2 -2692.063} C_VEL
LIN {X 0,Y 566.147,Z 744.032,A -85,B 0,C 180,E1 -2692.779,E2 -2692.779} C_VEL
LIN {X 0,Y 566.073,Z 752.523,A -85,B 0,C 180,E1 -2693.584,E2 -2693.584} C_VEL
LIN {X 0,Y 565.989,Z 759.932,A -85,B 0,C 180,E1 -2694.478,E2 -2694.478} C_VEL
LIN {X 0,Y 566.015,Z 765.662,A -85,B 0,C 180,E1 -2695.371,E2 -2695.371} C_VEL
LIN {X 0,Y 565.957,Z 770.842,A -85,B 0,C 180,E1 -2696.44,E2 -2696.44} C_VEL
LIN {X 0,Y 565.89,Z 773.443,A -85,B 0,C 180,E1 -2697.153,E2 -2697.153} C_VEL
LIN {X 0,Y 565.837,Z 775.411,A -85,B 0,C 180,E1 -2697.865,E2 -2697.865} C_VEL
LIN {X 0,Y 565.841,Z 776.833,A -85,B 0,C 180,E1 -2698.577,E2 -2698.577} C_VEL
LIN {X 0,Y 565.836,Z 777.689,A -85,B 0,C 180,E1 -2699.288,E2 -2699.288} C_VEL
LIN {X 0,Y 565.837,Z 777.996,A -85,B 0,C 180,E1 -2700,E2 -2700} C_VEL
LIN {X 0,Y 565.838,Z 777.756,A -85,B 0,C 180,E1 -2700.712,E2 -2700.712} C_VEL
LIN {X 0,Y 565.845,Z 776.967,A -85,B 0,C 180,E1 -2701.423,E2 -2701.423} C_VEL
LIN {X 0,Y 565.836,Z 775.614,A -85,B 0,C 180,E1 -2702.135,E2 -2702.135} C_VEL
LIN {X 0,Y 565.915,Z 772.571,A -85,B 0,C 180,E1 -2703.204,E2 -2703.204} C_VEL
LIN {X 0,Y 565.971,Z 768.029,A -85,B 0,C 180,E1 -2704.273,E2 -2704.273} C_VEL
LIN {X 0,Y 565.935,Z 762.951,A -85,B 0,C 180,E1 -2705.166,E2 -2705.166} C_VEL
LIN {X 0,Y 566.086,Z 756.465,A -85,B 0,C 180,E1 -2706.058,E2 -2706.058} C_VEL
LIN {X 0,Y 566.107,Z 748.039,A -85,B 0,C 180,E1 -2706.958,E2 -2706.958} C_VEL
LIN {X 0,Y 566.196,Z 739.424,A -85,B 0,C 180,E1 -2707.668,E2 -2707.668} C_VEL
LIN {X 0,Y 566.302,Z 729.683,A -85,B 0,C 180,E1 -2708.295,E2 -2708.295} C_VEL
LIN {X 0,Y 566.398,Z 719.25,A -85,B 0,C 180,E1 -2708.788,E2 -2708.788} C_VEL
LIN {X 0,Y 566.431,Z 709.138,A -85,B 0,C 180,E1 -2709.125,E2 -2709.125} C_VEL
LIN {X 0,Y 566.475,Z 698.378,A -85,B 0,C 180,E1 -2709.349,E2 -2709.349} C_VEL
LIN {X 0,Y 566.498,Z 634.211,A -85,B 0,C 180,E1 -2710.16,E2 -2710.16} C_VEL
LIN {X 0,Y 566.225,Z 630.98,A -85,B 0,C 180,E1 -2710.233,E2 -2710.233} C_VEL
LIN {X 0,Y 566.402,Z 607.054,A -85,B 0,C 180,E1 -2713.271,E2 -2713.271} C_VEL
LIN {X 0,Y 566.642,Z 584.313,A -85,B 0,C 180,E1 -2716.205,E2 -2716.205} C_VEL
LIN {X 0,Y 566.655,Z 580.776,A -85,B 0,C 180,E1 -2716.665,E2 -2716.665} C_VEL
LIN {X 0,Y 566.088,Z 577.263,A -85,B 0,C 180,E1 -2717.142,E2 -2717.142} C_VEL
LIN {X 0,Y 560.553,Z 566.501,A -85,B 0,C 180,E1 -2718.746,E2 -2718.746} C_VEL
LIN {X 0,Y 559.945,Z 563.017,A -85,B 0,C 180,E1 -2719.233,E2 -2719.233} C_VEL
LIN {X 0,Y 560.346,Z 540.182,A -85,B 0,C 180,E1 -2722.297,E2 -2722.297} C_VEL
LIN {X 0,Y 560.56,Z 522.55,A -85,B 0,C 180,E1 -2724.637,E2 -2724.637} C_VEL
LIN {X 0,Y 559.207,Z 514.909,A -85,B 0,C 180,E1 -2725.72,E2 -2725.72} C_VEL
LIN {X 0,Y 559.167,Z 514.836,A -85,B 0,C 180,E1 -2728.53,E2 -2728.53} C_VEL
LIN {X 0,Y 559.15,Z 514.83,A -85,B 0,C 180,E1 -2731.273,E2 -2731.273} C_VEL
LIN {X 0,Y 559.172,Z 514.83,A -85,B 0,C 180,E1 -2733.949,E2 -2733.949} C_VEL
LIN {X 0,Y 559.195,Z 514.834,A -85,B 0,C 180,E1 -2736.451,E2 -2736.451} C_VEL
LIN {X 0,Y 559.182,Z 514.828,A -85,B 0,C 180,E1 -2738.934,E2 -2738.934} C_VEL
LIN {X 0,Y 559.169,Z 514.823,A -85,B 0,C 180,E1 -2741.77,E2 -2741.77} C_VEL
LIN {X 0,Y 559.144,Z 514.836,A -85,B 0,C 180,E1 -2744.739,E2 -2744.739} C_VEL
LIN {X 0,Y 559.169,Z 514.828,A -85,B 0,C 180,E1 -2747.257,E2 -2747.257} C_VEL
LIN {X 0,Y 559.188,Z 514.825,A -85,B 0,C 180,E1 -2750.135,E2 -2750.135} C_VEL
LIN {X 0,Y 559.145,Z 514.835,A -85,B 0,C 180,E1 -2752.891,E2 -2752.891} C_VEL
LIN {X 0,Y 559.171,Z 514.827,A -85,B 0,C 180,E1 -2756.051,E2 -2756.051} C_VEL
LIN {X 0,Y 559.163,Z 514.832,A -85,B 0,C 180,E1 -2758.981,E2 -2758.981} C_VEL
LIN {X 0,Y 559.173,Z 514.826,A -85,B 0,C 180,E1 -2761.619,E2 -2761.619} C_VEL
LIN {X 0,Y 559.185,Z 514.826,A -85,B 0,C 180,E1 -2763.903,E2 -2763.903} C_VEL
LIN {X 0,Y 559.152,Z 514.835,A -85,B 0,C 180,E1 -2766.57,E2 -2766.57} C_VEL
LIN {X 0,Y 559.187,Z 514.831,A -85,B 0,C 180,E1 -2769.395,E2 -2769.395} C_VEL
LIN {X 0,Y 559.235,Z 514.989,A -85,B 0,C 180,E1 -2770.069,E2 -2770.069} C_VEL
LIN {X 0,Y 559.557,Z 520.655,A -85,B 0,C 180,E1 -2771.13,E2 -2771.13} C_VEL
LIN {X 0,Y 559.367,Z 536.379,A -85,B 0,C 180,E1 -2773.953,E2 -2773.953} C_VEL
LIN {X 0,Y 559.264,Z 547.229,A -85,B 0,C 180,E1 -2775.838,E2 -2775.838} C_VEL
LIN {X 0,Y 559.841,Z 550.889,A -85,B 0,C 180,E1 -2775.937,E2 -2775.937} C_VEL
LIN {X 0,Y 560.304,Z 554.745,A -85,B 0,C 180,E1 -2775.999,E2 -2775.999} C_VEL
LIN {X 0,Y 560.052,Z 653.971,A -85,B 0,C 180,E1 -2777.291,E2 -2777.291} C_VEL
LIN {X 0,Y 559.922,Z 667.237,A -85,B 0,C 180,E1 -2777.61,E2 -2777.61} C_VEL
LIN {X 0,Y 559.8,Z 679.391,A -85,B 0,C 180,E1 -2778.044,E2 -2778.044} C_VEL
LIN {X 0,Y 559.65,Z 691.07,A -85,B 0,C 180,E1 -2778.606,E2 -2778.606} C_VEL
LIN {X 0,Y 559.486,Z 702.558,A -85,B 0,C 180,E1 -2779.322,E2 -2779.322} C_VEL
LIN {X 0,Y 559.306,Z 713.073,A -85,B 0,C 180,E1 -2780.141,E2 -2780.141} C_VEL
LIN {X 0,Y 559.197,Z 721.671,A -85,B 0,C 180,E1 -2780.961,E2 -2780.961} C_VEL
LIN {X 0,Y 559.051,Z 729.591,A -85,B 0,C 180,E1 -2781.869,E2 -2781.869} C_VEL
LIN {X 0,Y 558.969,Z 737.451,A -85,B 0,C 180,E1 -2782.976,E2 -2782.976} C_VEL
LIN {X 0,Y 558.936,Z 744.452,A -85,B 0,C 180,E1 -2784.226,E2 -2784.226} C_VEL
LIN {X 0,Y 558.826,Z 749.194,A -85,B 0,C 180,E1 -2785.31,E2 -2785.31} C_VEL
LIN {X 0,Y 558.836,Z 752.826,A -85,B 0,C 180,E1 -2786.394,E2 -2786.394} C_VEL
LIN {X 0,Y 558.799,Z 754.703,A -85,B 0,C 180,E1 -2787.116,E2 -2787.116} C_VEL
LIN {X 0,Y 558.746,Z 756.128,A -85,B 0,C 180,E1 -2787.837,E2 -2787.837} C_VEL
LIN {X 0,Y 558.741,Z 757.756,A -85,B 0,C 180,E1 -2789.279,E2 -2789.279} C_VEL
LIN {X 0,Y 558.74,Z 757.996,A -85,B 0,C 180,E1 -2789.999,E2 -2789.999} C_VEL
LIN {X 0,Y 558.741,Z 757.815,A -85,B 0,C 180,E1 -2790.72,E2 -2790.72} C_VEL
LIN {X 0,Y 558.746,Z 756.27,A -85,B 0,C 180,E1 -2792.162,E2 -2792.162} C_VEL
LIN {X 0,Y 558.8,Z 754.909,A -85,B 0,C 180,E1 -2792.883,E2 -2792.883} C_VEL
LIN {X 0,Y 558.844,Z 752.03,A -85,B 0,C 180,E1 -2793.966,E2 -2793.966} C_VEL
LIN {X 0,Y 558.798,Z 748.129,A -85,B 0,C 180,E1 -2795.05,E2 -2795.05} C_VEL
LIN {X 0,Y 558.909,Z 743.097,A -85,B 0,C 180,E1 -2796.135,E2 -2796.135} C_VEL
LIN {X 0,Y 558.972,Z 736.773,A -85,B 0,C 180,E1 -2797.222,E2 -2797.222} C_VEL
LIN {X 0,Y 559.096,Z 728.85,A -85,B 0,C 180,E1 -2798.311,E2 -2798.311} C_VEL
LIN {X 0,Y 559.223,Z 718.998,A -85,B 0,C 180,E1 -2799.402,E2 -2799.402} C_VEL
LIN {X 0,Y 559.416,Z 708.682,A -85,B 0,C 180,E1 -2800.312,E2 -2800.312} C_VEL
LIN {X 0,Y 559.578,Z 697.759,A -85,B 0,C 180,E1 -2801.087,E2 -2801.087} C_VEL
LIN {X 0,Y 559.723,Z 686.188,A -85,B 0,C 180,E1 -2801.738,E2 -2801.738} C_VEL
LIN {X 0,Y 559.881,Z 673.604,A -85,B 0,C 180,E1 -2802.27,E2 -2802.27} C_VEL
LIN {X 0,Y 560.018,Z 660.428,A -85,B 0,C 180,E1 -2802.663,E2 -2802.663} C_VEL
LIN {X 0,Y 560.1,Z 648.06,A -85,B 0,C 180,E1 -2802.891,E2 -2802.891} C_VEL
LIN {X 0,Y 560.168,Z 552.704,A -85,B 0,C 180,E1 -2804.121,E2 -2804.121} C_VEL
LIN {X 0,Y 559.282,Z 547.55,A -85,B 0,C 180,E1 -2804.23,E2 -2804.23} C_VEL
LIN {X 0,Y 559.231,Z 546.34,A -85,B 0,C 180,E1 -2804.37,E2 -2804.37} C_VEL
LIN {X 0,Y 559.443,Z 529.865,A -85,B 0,C 180,E1 -2807.301,E2 -2807.301} C_VEL
LIN {X 0,Y 559.542,Z 517.108,A -85,B 0,C 180,E1 -2809.605,E2 -2809.605} C_VEL
LIN {X 0,Y 559.217,Z 514.889,A -85,B 0,C 180,E1 -2810.074,E2 -2810.074} C_VEL
LIN {X 0,Y 559.133,Z 514.837,A -85,B 0,C 180,E1 -2812.932,E2 -2812.932} C_VEL
LIN {X 0,Y 559.177,Z 514.835,A -85,B 0,C 180,E1 -2815.297,E2 -2815.297} C_VEL
LIN {X 0,Y 559.189,Z 514.829,A -85,B 0,C 180,E1 -2817.711,E2 -2817.711} C_VEL
LIN {X 0,Y 559.156,Z 514.828,A -85,B 0,C 180,E1 -2820.182,E2 -2820.182} C_VEL
LIN {X 0,Y 559.175,Z 514.827,A -85,B 0,C 180,E1 -2822.713,E2 -2822.713} C_VEL
LIN {X 0,Y 559.156,Z 514.838,A -85,B 0,C 180,E1 -2825.321,E2 -2825.321} C_VEL
LIN {X 0,Y 559.134,Z 514.833,A -85,B 0,C 180,E1 -2828.016,E2 -2828.016} C_VEL
LIN {X 0,Y 559.174,Z 514.826,A -85,B 0,C 180,E1 -2830.81,E2 -2830.81} C_VEL
LIN {X 0,Y 559.16,Z 514.831,A -85,B 0,C 180,E1 -2833.731,E2 -2833.731} C_VEL
LIN {X 0,Y 559.142,Z 514.831,A -85,B 0,C 180,E1 -2836.803,E2 -2836.803} C_VEL
LIN {X 0,Y 559.173,Z 514.832,A -85,B 0,C 180,E1 -2839.189,E2 -2839.189} C_VEL
LIN {X 0,Y 559.131,Z 514.831,A -85,B 0,C 180,E1 -2841.982,E2 -2841.982} C_VEL
LIN {X 0,Y 559.154,Z 514.829,A -85,B 0,C 180,E1 -2844.678,E2 -2844.678} C_VEL
LIN {X 0,Y 559.17,Z 514.835,A -85,B 0,C 180,E1 -2847.361,E2 -2847.361} C_VEL
LIN {X 0,Y 559.184,Z 514.826,A -85,B 0,C 180,E1 -2850.134,E2 -2850.134} C_VEL
LIN {X 0,Y 559.177,Z 514.829,A -85,B 0,C 180,E1 -2853.169,E2 -2853.169} C_VEL
LIN {X 0,Y 559.152,Z 514.839,A -85,B 0,C 180,E1 -2855.494,E2 -2855.494} C_VEL
LIN {X 0,Y 559.171,Z 514.825,A -85,B 0,C 180,E1 -2858.624,E2 -2858.624} C_VEL
LIN {X 0,Y 559.166,Z 514.829,A -85,B 0,C 180,E1 -2860.926,E2 -2860.926} C_VEL
LIN {X 0,Y 559.165,Z 514.829,A -85,B 0,C 180,E1 -2863.948,E2 -2863.948} C_VEL
LIN {X 0,Y 559.166,Z 514.828,A -85,B 0,C 180,E1 -2866.184,E2 -2866.184} C_VEL
LIN {X 0,Y 559.189,Z 514.827,A -85,B 0,C 180,E1 -2869.133,E2 -2869.133} C_VEL
LIN {X 0,Y 559.202,Z 514.825,A -85,B 0,C 180,E1 -2872.054,E2 -2872.054} C_VEL
LIN {X 0,Y 559.252,Z 514.818,A -85,B 0,C 180,E1 -2874.953,E2 -2874.953} C_VEL
LIN {X 0,Y 559.245,Z 514.822,A -85,B 0,C 180,E1 -2877.839,E2 -2877.839} C_VEL
LIN {X 0,Y 559.269,Z 514.814,A -85,B 0,C 180,E1 -2880.72,E2 -2880.72} C_VEL
LIN {X 0,Y 559.238,Z 514.818,A -85,B 0,C 180,E1 -2882.881,E2 -2882.881} C_VEL
LIN {X 0,Y 559.222,Z 514.827,A -85,B 0,C 180,E1 -2885.77,E2 -2885.77} C_VEL
LIN {X 0,Y 559.186,Z 514.824,A -85,B 0,C 180,E1 -2888.674,E2 -2888.674} C_VEL
LIN {X 0,Y 559.198,Z 514.832,A -85,B 0,C 180,E1 -2891.601,E2 -2891.601} C_VEL
LIN {X 0,Y 559.192,Z 514.823,A -85,B 0,C 180,E1 -2894.596,E2 -2894.596} C_VEL
LIN {X 0,Y 559.157,Z 514.836,A -85,B 0,C 180,E1 -2897.557,E2 -2897.557} C_VEL
LIN {X 0,Y 559.168,Z 514.833,A -85,B 0,C 180,E1 -2899.838,E2 -2899.838} C_VEL
LIN {X 0,Y 559.136,Z 514.832,A -85,B 0,C 180,E1 -2902.153,E2 -2902.153} C_VEL
LIN {X 0,Y 559.173,Z 514.83,A -85,B 0,C 180,E1 -2905.188,E2 -2905.188} C_VEL
LIN {X 0,Y 559.188,Z 514.833,A -85,B 0,C 180,E1 -2907.712,E2 -2907.712} C_VEL
LIN {X 0,Y 559.157,Z 514.829,A -85,B 0,C 180,E1 -2911.019,E2 -2911.019} C_VEL
LIN {X 0,Y 559.173,Z 514.831,A -85,B 0,C 180,E1 -2913.952,E2 -2913.952} C_VEL
LIN {X 0,Y 559.164,Z 514.824,A -85,B 0,C 180,E1 -2916.449,E2 -2916.449} C_VEL
LIN {X 0,Y 559.173,Z 514.827,A -85,B 0,C 180,E1 -2918.934,E2 -2918.934} C_VEL
LIN {X 0,Y 559.187,Z 514.83,A -85,B 0,C 180,E1 -2921.768,E2 -2921.768} C_VEL
LIN {X 0,Y 559.135,Z 514.831,A -85,B 0,C 180,E1 -2924.74,E2 -2924.74} C_VEL
LIN {X 0,Y 559.164,Z 514.829,A -85,B 0,C 180,E1 -2927.258,E2 -2927.258} C_VEL
LIN {X 0,Y 559.183,Z 514.827,A -85,B 0,C 180,E1 -2930.136,E2 -2930.136} C_VEL
LIN {X 0,Y 559.143,Z 514.827,A -85,B 0,C 180,E1 -2932.893,E2 -2932.893} C_VEL
LIN {X 0,Y 559.164,Z 514.83,A -85,B 0,C 180,E1 -2936.052,E2 -2936.052} C_VEL
LIN {X 0,Y 559.162,Z 514.813,A -85,B 0,C 180,E1 -2938.982,E2 -2938.982} C_VEL
LIN {X 0,Y 559.192,Z 514.825,A -85,B 0,C 180,E1 -2942.289,E2 -2942.289} C_VEL
LIN {X 0,Y 559.179,Z 514.828,A -85,B 0,C 180,E1 -2944.814,E2 -2944.814} C_VEL
LIN {X 0,Y 559.206,Z 515.04,A -85,B 0,C 180,E1 -2946.607,E2 -2946.607} C_VEL
LIN {X 0,Y 560.178,Z 520.515,A -85,B 0,C 180,E1 -2947.503,E2 -2947.503} C_VEL
LIN {X 0,Y 559.837,Z 539.746,A -85,B 0,C 180,E1 -2950.426,E2 -2950.426} C_VEL
LIN {X 0,Y 559.56,Z 558.324,A -85,B 0,C 180,E1 -2953.21,E2 -2953.21} C_VEL
LIN {X 0,Y 559.391,Z 576.037,A -85,B 0,C 180,E1 -2955.796,E2 -2955.796} C_VEL
LIN {X 0,Y 560.307,Z 583.356,A -85,B 0,C 180,E1 -2955.936,E2 -2955.936} C_VEL
LIN {X 0,Y 560.066,Z 683.982,A -85,B 0,C 180,E1 -2957.246,E2 -2957.246} C_VEL
LIN {X 0,Y 559.937,Z 696.475,A -85,B 0,C 180,E1 -2957.543,E2 -2957.543} C_VEL
LIN {X 0,Y 559.818,Z 709.389,A -85,B 0,C 180,E1 -2958,E2 -2958} C_VEL
LIN {X 0,Y 559.667,Z 720.825,A -85,B 0,C 180,E1 -2958.548,E2 -2958.548} C_VEL
LIN {X 0,Y 559.507,Z 731.919,A -85,B 0,C 180,E1 -2959.232,E2 -2959.232} C_VEL
LIN {X 0,Y 559.309,Z 742.548,A -85,B 0,C 180,E1 -2960.051,E2 -2960.051} C_VEL
LIN {X 0,Y 559.161,Z 752.12,A -85,B 0,C 180,E1 -2960.962,E2 -2960.962} C_VEL
LIN {X 0,Y 559.049,Z 759.966,A -85,B 0,C 180,E1 -2961.87,E2 -2961.87} C_VEL
LIN {X 0,Y 558.943,Z 767.627,A -85,B 0,C 180,E1 -2962.959,E2 -2962.959} C_VEL
LIN {X 0,Y 558.935,Z 774.683,A -85,B 0,C 180,E1 -2964.227,E2 -2964.227} C_VEL
LIN {X 0,Y 558.827,Z 779.374,A -85,B 0,C 180,E1 -2965.312,E2 -2965.312} C_VEL
LIN {X 0,Y 558.836,Z 782.961,A -85,B 0,C 180,E1 -2966.396,E2 -2966.396} C_VEL
LIN {X 0,Y 558.799,Z 784.811,A -85,B 0,C 180,E1 -2967.117,E2 -2967.117} C_VEL
LIN {X 0,Y 558.745,Z 787.187,A -85,B 0,C 180,E1 -2968.559,E2 -2968.559} C_VEL
LIN {X 0,Y 558.74,Z 788,A -85,B 0,C 180,E1 -2970.001,E2 -2970.001} C_VEL
LIN {X 0,Y 558.745,Z 787.184,A -85,B 0,C 180,E1 -2971.442,E2 -2971.442} C_VEL
LIN {X 0,Y 558.799,Z 784.806,A -85,B 0,C 180,E1 -2972.884,E2 -2972.884} C_VEL
LIN {X 0,Y 558.844,Z 781.893,A -85,B 0,C 180,E1 -2973.967,E2 -2973.967} C_VEL
LIN {X 0,Y 558.799,Z 777.947,A -85,B 0,C 180,E1 -2975.051,E2 -2975.051} C_VEL
LIN {X 0,Y 558.921,Z 772.864,A -85,B 0,C 180,E1 -2976.136,E2 -2976.136} C_VEL
LIN {X 0,Y 558.978,Z 766.464,A -85,B 0,C 180,E1 -2977.223,E2 -2977.223} C_VEL
LIN {X 0,Y 559.099,Z 758.473,A -85,B 0,C 180,E1 -2978.312,E2 -2978.312} C_VEL
LIN {X 0,Y 559.185,Z 750.329,A -85,B 0,C 180,E1 -2979.222,E2 -2979.222} C_VEL
LIN {X 0,Y 559.34,Z 740.394,A -85,B 0,C 180,E1 -2980.132,E2 -2980.132} C_VEL
LIN {X 0,Y 559.53,Z 729.387,A -85,B 0,C 180,E1 -2980.938,E2 -2980.938} C_VEL
LIN {X 0,Y 559.673,Z 717.451,A -85,B 0,C 180,E1 -2981.628,E2 -2981.628} C_VEL
LIN {X 0,Y 559.842,Z 704.758,A -85,B 0,C 180,E1 -2982.185,E2 -2982.185} C_VEL
LIN {X 0,Y 559.998,Z 691.33,A -85,B 0,C 180,E1 -2982.595,E2 -2982.595} C_VEL
LIN {X 0,Y 560.087,Z 678.043,A -85,B 0,C 180,E1 -2982.847,E2 -2982.847} C_VEL
LIN {X 0,Y 560.191,Z 581.365,A -85,B 0,C 180,E1 -2984.093,E2 -2984.093} C_VEL
LIN {X 0,Y 559.395,Z 576.017,A -85,B 0,C 180,E1 -2984.205,E2 -2984.205} C_VEL
LIN {X 0,Y 559.606,Z 556.399,A -85,B 0,C 180,E1 -2987.076,E2 -2987.076} C_VEL
LIN {X 0,Y 559.918,Z 536.907,A -85,B 0,C 180,E1 -2990.002,E2 -2990.002} C_VEL
LIN {X 0,Y 560.149,Z 520.503,A -85,B 0,C 180,E1 -2992.5,E2 -2992.5} C_VEL
LIN {X 0,Y 559.157,Z 514.913,A -85,B 0,C 180,E1 -2993.432,E2 -2993.432} C_VEL
LIN {X 0,Y 559.183,Z 514.829,A -85,B 0,C 180,E1 -2996.097,E2 -2996.097} C_VEL
LIN {X 0,Y 559.144,Z 514.827,A -85,B 0,C 180,E1 -2998.531,E2 -2998.531} C_VEL
LIN {X 0,Y 559.15,Z 514.831,A -85,B 0,C 180,E1 -3001.273,E2 -3001.273} C_VEL
LIN {X 0,Y 559.17,Z 514.835,A -85,B 0,C 180,E1 -3003.949,E2 -3003.949} C_VEL
LIN {X 0,Y 559.145,Z 514.83,A -85,B 0,C 180,E1 -3007.109,E2 -3007.109} C_VEL
LIN {X 0,Y 559.166,Z 514.836,A -85,B 0,C 180,E1 -3009.942,E2 -3009.942} C_VEL
LIN {X 0,Y 559.168,Z 514.828,A -85,B 0,C 180,E1 -3012.743,E2 -3012.743} C_VEL
LIN {X 0,Y 559.157,Z 514.836,A -85,B 0,C 180,E1 -3015.761,E2 -3015.761} C_VEL
LIN {X 0,Y 559.195,Z 514.83,A -85,B 0,C 180,E1 -3018.233,E2 -3018.233} C_VEL
LIN {X 0,Y 559.182,Z 514.827,A -85,B 0,C 180,E1 -3021.191,E2 -3021.191} C_VEL
LIN {X 0,Y 559.177,Z 514.835,A -85,B 0,C 180,E1 -3023.792,E2 -3023.792} C_VEL
LIN {X 0,Y 559.169,Z 514.83,A -85,B 0,C 180,E1 -3026.425,E2 -3026.425} C_VEL
LIN {X 0,Y 559.159,Z 514.83,A -85,B 0,C 180,E1 -3028.981,E2 -3028.981} C_VEL
LIN {X 0,Y 559.172,Z 514.836,A -85,B 0,C 180,E1 -3031.619,E2 -3031.619} C_VEL
LIN {X 0,Y 559.206,Z 514.942,A -85,B 0,C 180,E1 -3034.504,E2 -3034.504} C_VEL
LIN {X 0,Y 560.407,Z 521.223,A -85,B 0,C 180,E1 -3035.356,E2 -3035.356} C_VEL
LIN {X 0,Y 560.375,Z 536.467,A -85,B 0,C 180,E1 -3037.316,E2 -3037.316} C_VEL
LIN {X 0,Y 560.05,Z 556.635,A -85,B 0,C 180,E1 -3040.004,E2 -3040.004} C_VEL
LIN {X 0,Y 559.716,Z 578.604,A -85,B 0,C 180,E1 -3042.925,E2 -3042.925} C_VEL
LIN {X 0,Y 559.457,Z 600.676,A -85,B 0,C 180,E1 -3045.82,E2 -3045.82} C_VEL
LIN {X 0,Y 559.179,Z 623.428,A -85,B 0,C 180,E1 -3048.769,E2 -3048.769} C_VEL
LIN {X 0,Y 559.185,Z 631.003,A -85,B 0,C 180,E1 -3049.729,E2 -3049.729} C_VEL
LIN {X 0,Y 559.583,Z 636.07,A -85,B 0,C 180,E1 -3049.827,E2 -3049.827} C_VEL
LIN {X 0,Y 559.459,Z 702.426,A -85,B 0,C 180,E1 -3050.692,E2 -3050.692} C_VEL
LIN {X 0,Y 559.419,Z 714.445,A -85,B 0,C 180,E1 -3051.011,E2 -3051.011} C_VEL
LIN {X 0,Y 559.338,Z 724.407,A -85,B 0,C 180,E1 -3051.419,E2 -3051.419} C_VEL
LIN {X 0,Y 559.204,Z 734.203,A -85,B 0,C 180,E1 -3051.963,E2 -3051.963} C_VEL
LIN {X 0,Y 559.084,Z 744.038,A -85,B 0,C 180,E1 -3052.688,E2 -3052.688} C_VEL
LIN {X 0,Y 558.999,Z 752.532,A -85,B 0,C 180,E1 -3053.503,E2 -3053.503} C_VEL
LIN {X 0,Y 558.928,Z 759.935,A -85,B 0,C 180,E1 -3054.408,E2 -3054.408} C_VEL
LIN {X 0,Y 558.947,Z 765.67,A -85,B 0,C 180,E1 -3055.312,E2 -3055.312} C_VEL
LIN {X 0,Y 558.864,Z 770.85,A -85,B 0,C 180,E1 -3056.395,E2 -3056.395} C_VEL
LIN {X 0,Y 558.813,Z 773.45,A -85,B 0,C 180,E1 -3057.116,E2 -3057.116} C_VEL
LIN {X 0,Y 558.744,Z 775.414,A -85,B 0,C 180,E1 -3057.837,E2 -3057.837} C_VEL
LIN {X 0,Y 558.741,Z 776.832,A -85,B 0,C 180,E1 -3058.559,E2 -3058.559} C_VEL
LIN {X 0,Y 558.736,Z 777.687,A -85,B 0,C 180,E1 -3059.279,E2 -3059.279} C_VEL
LIN {X 0,Y 558.738,Z 777.996,A -85,B 0,C 180,E1 -3060,E2 -3060} C_VEL
LIN {X 0,Y 558.739,Z 777.758,A -85,B 0,C 180,E1 -3060.721,E2 -3060.721} C_VEL
LIN {X 0,Y 558.745,Z 776.97,A -85,B 0,C 180,E1 -3061.442,E2 -3061.442} C_VEL
LIN {X 0,Y 558.743,Z 775.616,A -85,B 0,C 180,E1 -3062.163,E2 -3062.163} C_VEL
LIN {X 0,Y 558.838,Z 772.566,A -85,B 0,C 180,E1 -3063.244,E2 -3063.244} C_VEL
LIN {X 0,Y 558.906,Z 768.025,A -85,B 0,C 180,E1 -3064.327,E2 -3064.327} C_VEL
LIN {X 0,Y 558.854,Z 762.953,A -85,B 0,C 180,E1 -3065.231,E2 -3065.231} C_VEL
LIN {X 0,Y 559.032,Z 756.467,A -85,B 0,C 180,E1 -3066.134,E2 -3066.134} C_VEL
LIN {X 0,Y 559.058,Z 748.275,A -85,B 0,C 180,E1 -3067.022,E2 -3067.022} C_VEL
LIN {X 0,Y 559.162,Z 739.424,A -85,B 0,C 180,E1 -3067.765,E2 -3067.765} C_VEL
LIN {X 0,Y 559.274,Z 729.675,A -85,B 0,C 180,E1 -3068.4,E2 -3068.4} C_VEL
LIN {X 0,Y 559.399,Z 719.239,A -85,B 0,C 180,E1 -3068.899,E2 -3068.899} C_VEL
LIN {X 0,Y 559.43,Z 708.292,A -85,B 0,C 180,E1 -3069.263,E2 -3069.263} C_VEL
LIN {X 0,Y 559.49,Z 696.779,A -85,B 0,C 180,E1 -3069.49,E2 -3069.49} C_VEL
LIN {X 0,Y 559.466,Z 634.165,A -85,B 0,C 180,E1 -3070.289,E2 -3070.289} C_VEL
LIN {X 0,Y 559.202,Z 630.977,A -85,B 0,C 180,E1 -3070.363,E2 -3070.363} C_VEL
LIN {X 0,Y 559.398,Z 605.628,A -85,B 0,C 180,E1 -3073.625,E2 -3073.625} C_VEL
LIN {X 0,Y 559.661,Z 584.309,A -85,B 0,C 180,E1 -3076.412,E2 -3076.412} C_VEL
LIN {X 0,Y 559.945,Z 563.017,A -85,B 0,C 180,E1 -3079.233,E2 -3079.233} C_VEL
LIN {X 0,Y 559.351,Z 559.584,A -85,B 0,C 180,E1 -3079.718,E2 -3079.718} C_VEL
LIN {X 0,Y 553.926,Z 548.893,A -85,B 0,C 180,E1 -3081.346,E2 -3081.346} C_VEL
LIN {X 0,Y 553.323,Z 545.346,A -85,B 0,C 180,E1 -3081.838,E2 -3081.838} C_VEL
LIN {X 0,Y 553.619,Z 524.967,A -85,B 0,C 180,E1 -3084.567,E2 -3084.567} C_VEL
LIN {X 0,Y 553.14,Z 520.667,A -85,B 0,C 180,E1 -3085.151,E2 -3085.151} C_VEL
LIN {X 0,Y 552.165,Z 515.794,A -85,B 0,C 180,E1 -3085.87,E2 -3085.87} C_VEL
LIN {X 0,Y 552.114,Z 515.71,A -85,B 0,C 180,E1 -3088.928,E2 -3088.928} C_VEL
LIN {X 0,Y 552.115,Z 515.707,A -85,B 0,C 180,E1 -3091.476,E2 -3091.476} C_VEL
LIN {X 0,Y 552.143,Z 515.708,A -85,B 0,C 180,E1 -3094.171,E2 -3094.171} C_VEL
LIN {X 0,Y 552.122,Z 515.71,A -85,B 0,C 180,E1 -3096.746,E2 -3096.746} C_VEL
LIN {X 0,Y 552.136,Z 515.702,A -85,B 0,C 180,E1 -3099.527,E2 -3099.527} C_VEL
LIN {X 0,Y 552.134,Z 515.704,A -85,B 0,C 180,E1 -3102.425,E2 -3102.425} C_VEL
LIN {X 0,Y 552.105,Z 515.706,A -85,B 0,C 180,E1 -3105.563,E2 -3105.563} C_VEL
LIN {X 0,Y 552.135,Z 515.708,A -85,B 0,C 180,E1 -3108.677,E2 -3108.677} C_VEL
LIN {X 0,Y 552.123,Z 515.702,A -85,B 0,C 180,E1 -3111.411,E2 -3111.411} C_VEL
LIN {X 0,Y 552.09,Z 515.712,A -85,B 0,C 180,E1 -3114.156,E2 -3114.156} C_VEL
LIN {X 0,Y 552.121,Z 515.712,A -85,B 0,C 180,E1 -3116.814,E2 -3116.814} C_VEL
LIN {X 0,Y 552.109,Z 515.707,A -85,B 0,C 180,E1 -3119.391,E2 -3119.391} C_VEL
LIN {X 0,Y 552.115,Z 515.706,A -85,B 0,C 180,E1 -3121.901,E2 -3121.901} C_VEL
LIN {X 0,Y 552.161,Z 515.709,A -85,B 0,C 180,E1 -3124.649,E2 -3124.649} C_VEL
LIN {X 0,Y 552.101,Z 515.709,A -85,B 0,C 180,E1 -3127.549,E2 -3127.549} C_VEL
LIN {X 0,Y 552.184,Z 515.887,A -85,B 0,C 180,E1 -3129.961,E2 -3129.961} C_VEL
LIN {X 0,Y 552.59,Z 520.659,A -85,B 0,C 180,E1 -3130.883,E2 -3130.883} C_VEL
LIN {X 0,Y 552.37,Z 535.334,A -85,B 0,C 180,E1 -3133.554,E2 -3133.554} C_VEL
LIN {X 0,Y 552.232,Z 547.195,A -85,B 0,C 180,E1 -3135.65,E2 -3135.65} C_VEL
LIN {X 0,Y 552.733,Z 550.374,A -85,B 0,C 180,E1 -3135.745,E2 -3135.745} C_VEL
LIN {X 0,Y 553.434,Z 555.043,A -85,B 0,C 180,E1 -3135.825,E2 -3135.825} C_VEL
LIN {X 0,Y 553.151,Z 654,A -85,B 0,C 180,E1 -3137.129,E2 -3137.129} C_VEL
LIN {X 0,Y 552.989,Z 667.256,A -85,B 0,C 180,E1 -3137.452,E2 -3137.452} C_VEL
LIN {X 0,Y 552.851,Z 679.398,A -85,B 0,C 180,E1 -3137.892,E2 -3137.892} C_VEL
LIN {X 0,Y 552.689,Z 690.893,A -85,B 0,C 180,E1 -3138.45,E2 -3138.45} C_VEL
LIN {X 0,Y 552.51,Z 702.564,A -85,B 0,C 180,E1 -3139.185,E2 -3139.185} C_VEL
LIN {X 0,Y 552.303,Z 713.081,A -85,B 0,C 180,E1 -3140.015,E2 -3140.015} C_VEL
LIN {X 0,Y 552.153,Z 721.677,A -85,B 0,C 180,E1 -3140.844,E2 -3140.844} C_VEL
LIN {X 0,Y 552.008,Z 729.596,A -85,B 0,C 180,E1 -3141.765,E2 -3141.765} C_VEL
LIN {X 0,Y 551.893,Z 737.455,A -85,B 0,C 180,E1 -3142.886,E2 -3142.886} C_VEL
LIN {X 0,Y 551.868,Z 744.455,A -85,B 0,C 180,E1 -3144.152,E2 -3144.152} C_VEL
LIN {X 0,Y 551.725,Z 749.196,A -85,B 0,C 180,E1 -3145.25,E2 -3145.25} C_VEL
LIN {X 0,Y 551.751,Z 752.828,A -85,B 0,C 180,E1 -3146.348,E2 -3146.348} C_VEL
LIN {X 0,Y 551.724,Z 754.705,A -85,B 0,C 180,E1 -3147.079,E2 -3147.079} C_VEL
LIN {X 0,Y 551.656,Z 756.129,A -85,B 0,C 180,E1 -3147.809,E2 -3147.809} C_VEL
LIN {X 0,Y 551.642,Z 757.756,A -85,B 0,C 180,E1 -3149.269,E2 -3149.269} C_VEL
LIN {X 0,Y 551.641,Z 757.996,A -85,B 0,C 180,E1 -3149.999,E2 -3149.999} C_VEL
LIN {X 0,Y 551.641,Z 757.815,A -85,B 0,C 180,E1 -3150.729,E2 -3150.729} C_VEL
LIN {X 0,Y 551.657,Z 756.269,A -85,B 0,C 180,E1 -3152.19,E2 -3152.19} C_VEL
LIN {X 0,Y 551.724,Z 754.908,A -85,B 0,C 180,E1 -3152.92,E2 -3152.92} C_VEL
LIN {X 0,Y 551.764,Z 752.028,A -85,B 0,C 180,E1 -3154.016,E2 -3154.016} C_VEL
LIN {X 0,Y 551.723,Z 748.127,A -85,B 0,C 180,E1 -3155.115,E2 -3155.115} C_VEL
LIN {X 0,Y 551.81,Z 742.398,A -85,B 0,C 180,E1 -3156.348,E2 -3156.348} C_VEL
LIN {X 0,Y 551.924,Z 735.542,A -85,B 0,C 180,E1 -3157.499,E2 -3157.499} C_VEL
LIN {X 0,Y 552.077,Z 727.358,A -85,B 0,C 180,E1 -3158.602,E2 -3158.602} C_VEL
LIN {X 0,Y 552.196,Z 718.992,A -85,B 0,C 180,E1 -3159.523,E2 -3159.523} C_VEL
LIN {X 0,Y 552.409,Z 708.676,A -85,B 0,C 180,E1 -3160.444,E2 -3160.444} C_VEL
LIN {X 0,Y 552.596,Z 698.044,A -85,B 0,C 180,E1 -3161.209,E2 -3161.209} C_VEL
LIN {X 0,Y 552.743,Z 687.274,A -85,B 0,C 180,E1 -3161.83,E2 -3161.83} C_VEL
LIN {X 0,Y 552.92,Z 674.754,A -85,B 0,C 180,E1 -3162.385,E2 -3162.385} C_VEL
LIN {X 0,Y 553.048,Z 661.322,A -85,B 0,C 180,E1 -3162.802,E2 -3162.802} C_VEL
LIN {X 0,Y 553.193,Z 648.018,A -85,B 0,C 180,E1 -3163.055,E2 -3163.055} C_VEL
LIN {X 0,Y 553.395,Z 554.455,A -85,B 0,C 180,E1 -3164.274,E2 -3164.274} C_VEL
LIN {X 0,Y 552.259,Z 547.491,A -85,B 0,C 180,E1 -3164.418,E2 -3164.418} C_VEL
LIN {X 0,Y 552.22,Z 545.276,A -85,B 0,C 180,E1 -3164.745,E2 -3164.745} C_VEL
LIN {X 0,Y 552.428,Z 530.477,A -85,B 0,C 180,E1 -3167.416,E2 -3167.416} C_VEL
LIN {X 0,Y 552.579,Z 518.47,A -85,B 0,C 180,E1 -3169.615,E2 -3169.615} C_VEL
LIN {X 0,Y 552.178,Z 515.759,A -85,B 0,C 180,E1 -3170.196,E2 -3170.196} C_VEL
LIN {X 0,Y 552.111,Z 515.715,A -85,B 0,C 180,E1 -3173.241,E2 -3173.241} C_VEL
LIN {X 0,Y 552.131,Z 515.708,A -85,B 0,C 180,E1 -3175.643,E2 -3175.643} C_VEL
LIN {X 0,Y 552.124,Z 515.705,A -85,B 0,C 180,E1 -3178.561,E2 -3178.561} C_VEL
LIN {X 0,Y 552.135,Z 515.712,A -85,B 0,C 180,E1 -3181.479,E2 -3181.479} C_VEL
LIN {X 0,Y 552.136,Z 515.704,A -85,B 0,C 180,E1 -3184.17,E2 -3184.17} C_VEL
LIN {X 0,Y 552.11,Z 515.706,A -85,B 0,C 180,E1 -3186.746,E2 -3186.746} C_VEL
LIN {X 0,Y 552.132,Z 515.71,A -85,B 0,C 180,E1 -3189.526,E2 -3189.526} C_VEL
LIN {X 0,Y 552.128,Z 515.704,A -85,B 0,C 180,E1 -3192.424,E2 -3192.424} C_VEL
LIN {X 0,Y 552.094,Z 515.715,A -85,B 0,C 180,E1 -3195.562,E2 -3195.562} C_VEL
LIN {X 0,Y 552.136,Z 515.703,A -85,B 0,C 180,E1 -3198.675,E2 -3198.675} C_VEL
LIN {X 0,Y 552.116,Z 515.71,A -85,B 0,C 180,E1 -3201.411,E2 -3201.411} C_VEL
LIN {X 0,Y 552.109,Z 515.707,A -85,B 0,C 180,E1 -3204.158,E2 -3204.158} C_VEL
LIN {X 0,Y 552.124,Z 515.705,A -85,B 0,C 180,E1 -3206.815,E2 -3206.815} C_VEL
LIN {X 0,Y 552.109,Z 515.714,A -85,B 0,C 180,E1 -3209.391,E2 -3209.391} C_VEL
LIN {X 0,Y 552.122,Z 515.706,A -85,B 0,C 180,E1 -3211.902,E2 -3211.902} C_VEL
LIN {X 0,Y 552.151,Z 515.701,A -85,B 0,C 180,E1 -3214.649,E2 -3214.649} C_VEL
LIN {X 0,Y 552.09,Z 515.716,A -85,B 0,C 180,E1 -3217.549,E2 -3217.549} C_VEL
LIN {X 0,Y 552.143,Z 515.702,A -85,B 0,C 180,E1 -3220.373,E2 -3220.373} C_VEL
LIN {X 0,Y 552.151,Z 515.702,A -85,B 0,C 180,E1 -3222.977,E2 -3222.977} C_VEL
LIN {X 0,Y 552.129,Z 515.706,A -85,B 0,C 180,E1 -3226.004,E2 -3226.004} C_VEL
LIN {X 0,Y 552.156,Z 515.702,A -85,B 0,C 180,E1 -3228.993,E2 -3228.993} C_VEL
LIN {X 0,Y 552.156,Z 515.704,A -85,B 0,C 180,E1 -3231.951,E2 -3231.951} C_VEL
LIN {X 0,Y 552.226,Z 515.693,A -85,B 0,C 180,E1 -3234.889,E2 -3234.889} C_VEL
LIN {X 0,Y 552.217,Z 515.698,A -85,B 0,C 180,E1 -3237.812,E2 -3237.812} C_VEL
LIN {X 0,Y 552.239,Z 515.69,A -85,B 0,C 180,E1 -3240.729,E2 -3240.729} C_VEL
LIN {X 0,Y 552.204,Z 515.694,A -85,B 0,C 180,E1 -3242.918,E2 -3242.918} C_VEL
LIN {X 0,Y 552.192,Z 515.701,A -85,B 0,C 180,E1 -3245.844,E2 -3245.844} C_VEL
LIN {X 0,Y 552.156,Z 515.7,A -85,B 0,C 180,E1 -3248.786,E2 -3248.786} C_VEL
LIN {X 0,Y 552.155,Z 515.708,A -85,B 0,C 180,E1 -3251.751,E2 -3251.751} C_VEL
LIN {X 0,Y 552.129,Z 515.703,A -85,B 0,C 180,E1 -3254.749,E2 -3254.749} C_VEL
LIN {X 0,Y 552.108,Z 515.713,A -85,B 0,C 180,E1 -3257.789,E2 -3257.789} C_VEL
LIN {X 0,Y 552.127,Z 515.706,A -85,B 0,C 180,E1 -3260.101,E2 -3260.101} C_VEL
LIN {X 0,Y 552.089,Z 515.708,A -85,B 0,C 180,E1 -3262.451,E2 -3262.451} C_VEL
LIN {X 0,Y 552.15,Z 515.707,A -85,B 0,C 180,E1 -3265.351,E2 -3265.351} C_VEL
LIN {X 0,Y 552.12,Z 515.708,A -85,B 0,C 180,E1 -3268.098,E2 -3268.098} C_VEL
LIN {X 0,Y 552.101,Z 515.706,A -85,B 0,C 180,E1 -3270.609,E2 -3270.609} C_VEL
LIN {X 0,Y 552.124,Z 515.708,A -85,B 0,C 180,E1 -3273.185,E2 -3273.185} C_VEL
LIN {X 0,Y 552.109,Z 515.709,A -85,B 0,C 180,E1 -3275.842,E2 -3275.842} C_VEL
LIN {X 0,Y 552.121,Z 515.706,A -85,B 0,C 180,E1 -3279.063,E2 -3279.063} C_VEL
LIN {X 0,Y 552.135,Z 515.709,A -85,B 0,C 180,E1 -3281.445,E2 -3281.445} C_VEL
LIN {X 0,Y 552.091,Z 515.709,A -85,B 0,C 180,E1 -3284.533,E2 -3284.533} C_VEL
LIN {X 0,Y 552.128,Z 515.711,A -85,B 0,C 180,E1 -3287.585,E2 -3287.585} C_VEL
LIN {X 0,Y 552.131,Z 515.702,A -85,B 0,C 180,E1 -3290.474,E2 -3290.474} C_VEL
LIN {X 0,Y 552.109,Z 515.706,A -85,B 0,C 180,E1 -3293.317,E2 -3293.317} C_VEL
LIN {X 0,Y 552.127,Z 515.708,A -85,B 0,C 180,E1 -3295.94,E2 -3295.94} C_VEL
LIN {X 0,Y 552.117,Z 515.689,A -85,B 0,C 180,E1 -3298.541,E2 -3298.541} C_VEL
LIN {X 0,Y 552.125,Z 515.71,A -85,B 0,C 180,E1 -3301.439,E2 -3301.439} C_VEL
LIN {X 0,Y 552.13,Z 515.702,A -85,B 0,C 180,E1 -3304.357,E2 -3304.357} C_VEL
LIN {X 0,Y 552.146,Z 515.888,A -85,B 0,C 180,E1 -3306.448,E2 -3306.448} C_VEL
LIN {X 0,Y 553.221,Z 521.628,A -85,B 0,C 180,E1 -3307.401,E2 -3307.401} C_VEL
LIN {X 0,Y 552.899,Z 541.412,A -85,B 0,C 180,E1 -3310.426,E2 -3310.426} C_VEL
LIN {X 0,Y 552.569,Z 559.584,A -85,B 0,C 180,E1 -3313.182,E2 -3313.182} C_VEL
LIN {X 0,Y 552.393,Z 575.99,A -85,B 0,C 180,E1 -3315.609,E2 -3315.609} C_VEL
LIN {X 0,Y 553.434,Z 583.83,A -85,B 0,C 180,E1 -3315.764,E2 -3315.764} C_VEL
LIN {X 0,Y 553.157,Z 683.982,A -85,B 0,C 180,E1 -3317.084,E2 -3317.084} C_VEL
LIN {X 0,Y 553.012,Z 697.235,A -85,B 0,C 180,E1 -3317.407,E2 -3317.407} C_VEL
LIN {X 0,Y 552.857,Z 709.382,A -85,B 0,C 180,E1 -3317.846,E2 -3317.846} C_VEL
LIN {X 0,Y 552.689,Z 721.677,A -85,B 0,C 180,E1 -3318.45,E2 -3318.45} C_VEL
LIN {X 0,Y 552.505,Z 733.209,A -85,B 0,C 180,E1 -3319.187,E2 -3319.187} C_VEL
LIN {X 0,Y 552.295,Z 743.611,A -85,B 0,C 180,E1 -3320.016,E2 -3320.016} C_VEL
LIN {X 0,Y 552.125,Z 752.12,A -85,B 0,C 180,E1 -3320.845,E2 -3320.845} C_VEL
LIN {X 0,Y 552.012,Z 759.966,A -85,B 0,C 180,E1 -3321.766,E2 -3321.766} C_VEL
LIN {X 0,Y 551.889,Z 767.626,A -85,B 0,C 180,E1 -3322.868,E2 -3322.868} C_VEL
LIN {X 0,Y 551.867,Z 774.683,A -85,B 0,C 180,E1 -3324.153,E2 -3324.153} C_VEL
LIN {X 0,Y 551.725,Z 779.374,A -85,B 0,C 180,E1 -3325.251,E2 -3325.251} C_VEL
LIN {X 0,Y 551.75,Z 782.962,A -85,B 0,C 180,E1 -3326.349,E2 -3326.349} C_VEL
LIN {X 0,Y 551.723,Z 784.811,A -85,B 0,C 180,E1 -3327.08,E2 -3327.08} C_VEL
LIN {X 0,Y 551.645,Z 787.186,A -85,B 0,C 180,E1 -3328.541,E2 -3328.541} C_VEL
LIN {X 0,Y 551.64,Z 788,A -85,B 0,C 180,E1 -3330.001,E2 -3330.001} C_VEL
LIN {X 0,Y 551.645,Z 787.184,A -85,B 0,C 180,E1 -3331.461,E2 -3331.461} C_VEL
LIN {X 0,Y 551.724,Z 784.806,A -85,B 0,C 180,E1 -3332.921,E2 -3332.921} C_VEL
LIN {X 0,Y 551.764,Z 781.893,A -85,B 0,C 180,E1 -3334.018,E2 -3334.018} C_VEL
LIN {X 0,Y 551.724,Z 777.947,A -85,B 0,C 180,E1 -3335.116,E2 -3335.116} C_VEL
LIN {X 0,Y 551.803,Z 772.189,A -85,B 0,C 180,E1 -3336.342,E2 -3336.342} C_VEL
LIN {X 0,Y 551.927,Z 765.232,A -85,B 0,C 180,E1 -3337.5,E2 -3337.5} C_VEL
LIN {X 0,Y 552.083,Z 756.986,A -85,B 0,C 180,E1 -3338.603,E2 -3338.603} C_VEL
LIN {X 0,Y 552.223,Z 748.533,A -85,B 0,C 180,E1 -3339.524,E2 -3339.524} C_VEL
LIN {X 0,Y 552.385,Z 738.088,A -85,B 0,C 180,E1 -3340.446,E2 -3340.446} C_VEL
LIN {X 0,Y 552.601,Z 727.277,A -85,B 0,C 180,E1 -3341.214,E2 -3341.214} C_VEL
LIN {X 0,Y 552.754,Z 716.398,A -85,B 0,C 180,E1 -3341.831,E2 -3341.831} C_VEL
LIN {X 0,Y 552.908,Z 704.756,A -85,B 0,C 180,E1 -3342.34,E2 -3342.34} C_VEL
LIN {X 0,Y 553.057,Z 691.329,A -85,B 0,C 180,E1 -3342.756,E2 -3342.756} C_VEL
LIN {X 0,Y 553.19,Z 678.043,A -85,B 0,C 180,E1 -3343.01,E2 -3343.01} C_VEL
LIN {X 0,Y 553.403,Z 582.637,A -85,B 0,C 180,E1 -3344.253,E2 -3344.253} C_VEL
LIN {X 0,Y 552.405,Z 575.972,A -85,B 0,C 180,E1 -3344.392,E2 -3344.392} C_VEL
LIN {X 0,Y 552.667,Z 555.091,A -85,B 0,C 180,E1 -3347.495,E2 -3347.495} C_VEL
LIN {X 0,Y 553.023,Z 534.355,A -85,B 0,C 180,E1 -3350.65,E2 -3350.65} C_VEL
LIN {X 0,Y 553.19,Z 521.605,A -85,B 0,C 180,E1 -3352.601,E2 -3352.601} C_VEL
LIN {X 0,Y 552.126,Z 515.83,A -85,B 0,C 180,E1 -3353.582,E2 -3353.582} C_VEL
LIN {X 0,Y 552.133,Z 515.704,A -85,B 0,C 180,E1 -3355.645,E2 -3355.645} C_VEL
LIN {X 0,Y 552.109,Z 515.702,A -85,B 0,C 180,E1 -3358.559,E2 -3358.559} C_VEL
LIN {X 0,Y 552.115,Z 515.708,A -85,B 0,C 180,E1 -3361.476,E2 -3361.476} C_VEL
LIN {X 0,Y 552.137,Z 515.713,A -85,B 0,C 180,E1 -3364.17,E2 -3364.17} C_VEL
LIN {X 0,Y 552.109,Z 515.708,A -85,B 0,C 180,E1 -3366.747,E2 -3366.747} C_VEL
LIN {X 0,Y 552.134,Z 515.706,A -85,B 0,C 180,E1 -3369.527,E2 -3369.527} C_VEL
LIN {X 0,Y 552.136,Z 515.707,A -85,B 0,C 180,E1 -3372.425,E2 -3372.425} C_VEL
LIN {X 0,Y 552.102,Z 515.712,A -85,B 0,C 180,E1 -3375.563,E2 -3375.563} C_VEL
LIN {X 0,Y 552.144,Z 515.704,A -85,B 0,C 180,E1 -3378.676,E2 -3378.676} C_VEL
LIN {X 0,Y 552.124,Z 515.708,A -85,B 0,C 180,E1 -3381.411,E2 -3381.411} C_VEL
LIN {X 0,Y 552.117,Z 515.711,A -85,B 0,C 180,E1 -3384.159,E2 -3384.159} C_VEL
LIN {X 0,Y 552.127,Z 515.706,A -85,B 0,C 180,E1 -3386.815,E2 -3386.815} C_VEL
LIN {X 0,Y 552.106,Z 515.712,A -85,B 0,C 180,E1 -3389.391,E2 -3389.391} C_VEL
LIN {X 0,Y 552.113,Z 515.715,A -85,B 0,C 180,E1 -3391.902,E2 -3391.902} C_VEL
LIN {X 0,Y 552.156,Z 515.885,A -85,B 0,C 180,E1 -3394.44,E2 -3394.44} C_VEL
LIN {X 0,Y 553.482,Z 523.257,A -85,B 0,C 180,E1 -3395.427,E2 -3395.427} C_VEL
LIN {X 0,Y 553.304,Z 544.106,A -85,B 0,C 180,E1 -3398.109,E2 -3398.109} C_VEL
LIN {X 0,Y 553.055,Z 563.743,A -85,B 0,C 180,E1 -3400.707,E2 -3400.707} C_VEL
LIN {X 0,Y 552.667,Z 586.473,A -85,B 0,C 180,E1 -3403.754,E2 -3403.754} C_VEL
LIN {X 0,Y 552.381,Z 607.784,A -85,B 0,C 180,E1 -3406.574,E2 -3406.574} C_VEL
LIN {X 0,Y 552.164,Z 631.016,A -85,B 0,C 180,E1 -3409.596,E2 -3409.596} C_VEL
LIN {X 0,Y 552.625,Z 637.904,A -85,B 0,C 180,E1 -3409.721,E2 -3409.721} C_VEL
LIN {X 0,Y 552.465,Z 702.45,A -85,B 0,C 180,E1 -3410.573,E2 -3410.573} C_VEL
LIN {X 0,Y 552.405,Z 714.457,A -85,B 0,C 180,E1 -3410.895,E2 -3410.895} C_VEL
LIN {X 0,Y 552.327,Z 724.432,A -85,B 0,C 180,E1 -3411.309,E2 -3411.309} C_VEL
LIN {X 0,Y 552.189,Z 734.221,A -85,B 0,C 180,E1 -3411.86,E2 -3411.86} C_VEL
LIN {X 0,Y 552.051,Z 744.043,A -85,B 0,C 180,E1 -3412.594,E2 -3412.594} C_VEL
LIN {X 0,Y 551.951,Z 752.54,A -85,B 0,C 180,E1 -3413.42,E2 -3413.42} C_VEL
LIN {X 0,Y 551.871,Z 759.938,A -85,B 0,C 180,E1 -3414.336,E2 -3414.336} C_VEL
LIN {X 0,Y 551.871,Z 765.677,A -85,B 0,C 180,E1 -3415.252,E2 -3415.252} C_VEL
LIN {X 0,Y 551.775,Z 770.857,A -85,B 0,C 180,E1 -3416.349,E2 -3416.349} C_VEL
LIN {X 0,Y 551.74,Z 773.458,A -85,B 0,C 180,E1 -3417.079,E2 -3417.079} C_VEL
LIN {X 0,Y 551.655,Z 775.418,A -85,B 0,C 180,E1 -3417.81,E2 -3417.81} C_VEL
LIN {X 0,Y 551.641,Z 776.83,A -85,B 0,C 180,E1 -3418.54,E2 -3418.54} C_VEL
LIN {X 0,Y 551.637,Z 777.685,A -85,B 0,C 180,E1 -3419.27,E2 -3419.27} C_VEL
LIN {X 0,Y 551.638,Z 777.996,A -85,B 0,C 180,E1 -3420,E2 -3420} C_VEL
LIN {X 0,Y 551.639,Z 777.759,A -85,B 0,C 180,E1 -3420.73,E2 -3420.73} C_VEL
LIN {X 0,Y 551.644,Z 776.97,A -85,B 0,C 180,E1 -3421.46,E2 -3421.46} C_VEL
LIN {X 0,Y 551.654,Z 775.617,A -85,B 0,C 180,E1 -3422.19,E2 -3422.19} C_VEL
LIN {X 0,Y 551.764,Z 772.561,A -85,B 0,C 180,E1 -3423.286,E2 -3423.286} C_VEL
LIN {X 0,Y 551.825,Z 768.022,A -85,B 0,C 180,E1 -3424.383,E2 -3424.383} C_VEL
LIN {X 0,Y 551.782,Z 762.954,A -85,B 0,C 180,E1 -3425.298,E2 -3425.298} C_VEL
LIN {X 0,Y 551.977,Z 756.687,A -85,B 0,C 180,E1 -3426.185,E2 -3426.185} C_VEL
LIN {X 0,Y 551.974,Z 749.961,A -85,B 0,C 180,E1 -3426.947,E2 -3426.947} C_VEL
LIN {X 0,Y 552.101,Z 740.623,A -85,B 0,C 180,E1 -3427.773,E2 -3427.773} C_VEL
LIN {X 0,Y 552.25,Z 731.191,A -85,B 0,C 180,E1 -3428.416,E2 -3428.416} C_VEL
LIN {X 0,Y 552.385,Z 720.384,A -85,B 0,C 180,E1 -3428.967,E2 -3428.967} C_VEL
LIN {X 0,Y 552.437,Z 709.134,A -85,B 0,C 180,E1 -3429.358,E2 -3429.358} C_VEL
LIN {X 0,Y 552.478,Z 698.301,A -85,B 0,C 180,E1 -3429.588,E2 -3429.588} C_VEL
LIN {X 0,Y 552.536,Z 635.016,A -85,B 0,C 180,E1 -3430.408,E2 -3430.408} C_VEL
LIN {X 0,Y 552.16,Z 630.975,A -85,B 0,C 180,E1 -3430.496,E2 -3430.496} C_VEL
LIN {X 0,Y 552.38,Z 607.044,A -85,B 0,C 180,E1 -3433.614,E2 -3433.614} C_VEL
LIN {X 0,Y 552.695,Z 584.304,A -85,B 0,C 180,E1 -3436.625,E2 -3436.625} C_VEL
LIN {X 0,Y 553.067,Z 562.265,A -85,B 0,C 180,E1 -3439.583,E2 -3439.583} C_VEL
LIN {X 0,Y 553.323,Z 545.346,A -85,B 0,C 180,E1 -3441.838,E2 -3441.838} C_VEL
LIN {X 0,Y 552.721,Z 541.847,A -85,B 0,C 180,E1 -3442.327,E2 -3442.327} C_VEL
LIN {X 0,Y 547.301,Z 531.09,A -85,B 0,C 180,E1 -3443.972,E2 -3443.972} C_VEL
LIN {X 0,Y 546.671,Z 527.559,A -85,B 0,C 180,E1 -3444.468,E2 -3444.468} C_VEL
LIN {X 0,Y 546.336,Z 522.77,A -85,B 0,C 180,E1 -3445.12,E2 -3445.12} C_VEL
LIN {X 0,Y 545.123,Z 516.674,A -85,B 0,C 180,E1 -3446.024,E2 -3446.024} C_VEL
LIN {X 0,Y 545.093,Z 516.587,A -85,B 0,C 180,E1 -3448.748,E2 -3448.748} C_VEL
LIN {X 0,Y 545.062,Z 516.586,A -85,B 0,C 180,E1 -3451.679,E2 -3451.679} C_VEL
LIN {X 0,Y 545.086,Z 516.59,A -85,B 0,C 180,E1 -3454.563,E2 -3454.563} C_VEL
LIN {X 0,Y 545.046,Z 516.587,A -85,B 0,C 180,E1 -3457.303,E2 -3457.303} C_VEL
LIN {X 0,Y 545.075,Z 516.586,A -85,B 0,C 180,E1 -3460.142,E2 -3460.142} C_VEL
LIN {X 0,Y 545.083,Z 516.576,A -85,B 0,C 180,E1 -3463.107,E2 -3463.107} C_VEL
LIN {X 0,Y 545.07,Z 516.587,A -85,B 0,C 180,E1 -3466.224,E2 -3466.224} C_VEL
LIN {X 0,Y 545.093,Z 516.581,A -85,B 0,C 180,E1 -3468.886,E2 -3468.886} C_VEL
LIN {X 0,Y 545.058,Z 516.582,A -85,B 0,C 180,E1 -3471.763,E2 -3471.763} C_VEL
LIN {X 0,Y 545.041,Z 516.596,A -85,B 0,C 180,E1 -3474.531,E2 -3474.531} C_VEL
LIN {X 0,Y 545.074,Z 516.585,A -85,B 0,C 180,E1 -3477.211,E2 -3477.211} C_VEL
LIN {X 0,Y 545.069,Z 516.584,A -85,B 0,C 180,E1 -3479.81,E2 -3479.81} C_VEL
LIN {X 0,Y 545.086,Z 516.586,A -85,B 0,C 180,E1 -3482.344,E2 -3482.344} C_VEL
LIN {X 0,Y 545.123,Z 516.582,A -85,B 0,C 180,E1 -3484.82,E2 -3484.82} C_VEL
LIN {X 0,Y 545.047,Z 516.589,A -85,B 0,C 180,E1 -3487.242,E2 -3487.242} C_VEL
LIN {X 0,Y 545.154,Z 516.754,A -85,B 0,C 180,E1 -3489.827,E2 -3489.827} C_VEL
LIN {X 0,Y 545.627,Z 521.841,A -85,B 0,C 180,E1 -3490.824,E2 -3490.824} C_VEL
LIN {X 0,Y 545.367,Z 536.385,A -85,B 0,C 180,E1 -3493.53,E2 -3493.53} C_VEL
LIN {X 0,Y 545.179,Z 546.321,A -85,B 0,C 180,E1 -3495.326,E2 -3495.326} C_VEL
LIN {X 0,Y 545.289,Z 548.011,A -85,B 0,C 180,E1 -3495.503,E2 -3495.503} C_VEL
LIN {X 0,Y 546.565,Z 555.587,A -85,B 0,C 180,E1 -3495.649,E2 -3495.649} C_VEL
LIN {X 0,Y 546.232,Z 654.029,A -85,B 0,C 180,E1 -3496.963,E2 -3496.963} C_VEL
LIN {X 0,Y 546.076,Z 667.275,A -85,B 0,C 180,E1 -3497.291,E2 -3497.291} C_VEL
LIN {X 0,Y 545.899,Z 679.414,A -85,B 0,C 180,E1 -3497.735,E2 -3497.735} C_VEL
LIN {X 0,Y 545.728,Z 691.607,A -85,B 0,C 180,E1 -3498.342,E2 -3498.342} C_VEL
LIN {X 0,Y 545.531,Z 702.571,A -85,B 0,C 180,E1 -3499.045,E2 -3499.045} C_VEL
LIN {X 0,Y 545.266,Z 713.087,A -85,B 0,C 180,E1 -3499.885,E2 -3499.885} C_VEL
LIN {X 0,Y 545.122,Z 721.683,A -85,B 0,C 180,E1 -3500.725,E2 -3500.725} C_VEL
LIN {X 0,Y 544.976,Z 729.601,A -85,B 0,C 180,E1 -3501.657,E2 -3501.657} C_VEL
LIN {X 0,Y 544.828,Z 737.347,A -85,B 0,C 180,E1 -3502.774,E2 -3502.774} C_VEL
LIN {X 0,Y 544.778,Z 744.458,A -85,B 0,C 180,E1 -3504.076,E2 -3504.076} C_VEL
LIN {X 0,Y 544.629,Z 749.199,A -85,B 0,C 180,E1 -3505.188,E2 -3505.188} C_VEL
LIN {X 0,Y 544.669,Z 752.83,A -85,B 0,C 180,E1 -3506.3,E2 -3506.3} C_VEL
LIN {X 0,Y 544.65,Z 754.707,A -85,B 0,C 180,E1 -3507.041,E2 -3507.041} C_VEL
LIN {X 0,Y 544.571,Z 756.129,A -85,B 0,C 180,E1 -3507.78,E2 -3507.78} C_VEL
LIN {X 0,Y 544.542,Z 757.757,A -85,B 0,C 180,E1 -3509.26,E2 -3509.26} C_VEL
LIN {X 0,Y 544.542,Z 757.996,A -85,B 0,C 180,E1 -3509.999,E2 -3509.999} C_VEL
LIN {X 0,Y 544.542,Z 757.815,A -85,B 0,C 180,E1 -3510.739,E2 -3510.739} C_VEL
LIN {X 0,Y 544.571,Z 756.268,A -85,B 0,C 180,E1 -3512.218,E2 -3512.218} C_VEL
LIN {X 0,Y 544.651,Z 754.906,A -85,B 0,C 180,E1 -3512.958,E2 -3512.958} C_VEL
LIN {X 0,Y 544.684,Z 752.026,A -85,B 0,C 180,E1 -3514.069,E2 -3514.069} C_VEL
LIN {X 0,Y 544.653,Z 748.125,A -85,B 0,C 180,E1 -3515.182,E2 -3515.182} C_VEL
LIN {X 0,Y 544.724,Z 742.9,A -85,B 0,C 180,E1 -3516.335,E2 -3516.335} C_VEL
LIN {X 0,Y 544.858,Z 735.538,A -85,B 0,C 180,E1 -3517.597,E2 -3517.597} C_VEL
LIN {X 0,Y 545.025,Z 727.353,A -85,B 0,C 180,E1 -3518.714,E2 -3518.714} C_VEL
LIN {X 0,Y 545.157,Z 718.986,A -85,B 0,C 180,E1 -3519.647,E2 -3519.647} C_VEL
LIN {X 0,Y 545.389,Z 708.667,A -85,B 0,C 180,E1 -3520.58,E2 -3520.58} C_VEL
LIN {X 0,Y 545.647,Z 697.333,A -85,B 0,C 180,E1 -3521.4,E2 -3521.4} C_VEL
LIN {X 0,Y 545.787,Z 687.261,A -85,B 0,C 180,E1 -3521.983,E2 -3521.983} C_VEL
LIN {X 0,Y 545.981,Z 674.739,A -85,B 0,C 180,E1 -3522.545,E2 -3522.545} C_VEL
LIN {X 0,Y 546.145,Z 661.298,A -85,B 0,C 180,E1 -3522.966,E2 -3522.966} C_VEL
LIN {X 0,Y 546.286,Z 647.976,A -85,B 0,C 180,E1 -3523.223,E2 -3523.223} C_VEL
LIN {X 0,Y 546.504,Z 555.031,A -85,B 0,C 180,E1 -3524.45,E2 -3524.45} C_VEL
LIN {X 0,Y 545.259,Z 547.716,A -85,B 0,C 180,E1 -3524.6,E2 -3524.6} C_VEL
LIN {X 0,Y 545.229,Z 545.273,A -85,B 0,C 180,E1 -3524.939,E2 -3524.939} C_VEL
LIN {X 0,Y 545.533,Z 528.563,A -85,B 0,C 180,E1 -3528.009,E2 -3528.009} C_VEL
LIN {X 0,Y 545.465,Z 518.774,A -85,B 0,C 180,E1 -3529.853,E2 -3529.853} C_VEL
LIN {X 0,Y 545.124,Z 516.676,A -85,B 0,C 180,E1 -3530.293,E2 -3530.293} C_VEL
LIN {X 0,Y 545.093,Z 516.587,A -85,B 0,C 180,E1 -3533.558,E2 -3533.558} C_VEL
LIN {X 0,Y 545.08,Z 516.583,A -85,B 0,C 180,E1 -3536,E2 -3536} C_VEL
LIN {X 0,Y 545.089,Z 516.582,A -85,B 0,C 180,E1 -3538.747,E2 -3538.747} C_VEL
LIN {X 0,Y 545.077,Z 516.588,A -85,B 0,C 180,E1 -3541.682,E2 -3541.682} C_VEL
LIN {X 0,Y 545.08,Z 516.583,A -85,B 0,C 180,E1 -3544.562,E2 -3544.562} C_VEL
LIN {X 0,Y 545.039,Z 516.594,A -85,B 0,C 180,E1 -3547.303,E2 -3547.303} C_VEL
LIN {X 0,Y 545.072,Z 516.582,A -85,B 0,C 180,E1 -3550.141,E2 -3550.141} C_VEL
LIN {X 0,Y 545.084,Z 516.586,A -85,B 0,C 180,E1 -3553.105,E2 -3553.105} C_VEL
LIN {X 0,Y 545.063,Z 516.584,A -85,B 0,C 180,E1 -3556.223,E2 -3556.223} C_VEL
LIN {X 0,Y 545.097,Z 516.582,A -85,B 0,C 180,E1 -3558.887,E2 -3558.887} C_VEL
LIN {X 0,Y 545.05,Z 516.587,A -85,B 0,C 180,E1 -3561.762,E2 -3561.762} C_VEL
LIN {X 0,Y 545.061,Z 516.584,A -85,B 0,C 180,E1 -3564.533,E2 -3564.533} C_VEL
LIN {X 0,Y 545.078,Z 516.588,A -85,B 0,C 180,E1 -3567.212,E2 -3567.212} C_VEL
LIN {X 0,Y 545.096,Z 516.584,A -85,B 0,C 180,E1 -3569.812,E2 -3569.812} C_VEL
LIN {X 0,Y 545.096,Z 516.579,A -85,B 0,C 180,E1 -3572.824,E2 -3572.824} C_VEL
LIN {X 0,Y 545.047,Z 516.593,A -85,B 0,C 180,E1 -3575.63,E2 -3575.63} C_VEL
LIN {X 0,Y 545.063,Z 516.583,A -85,B 0,C 180,E1 -3578.836,E2 -3578.836} C_VEL
LIN {X 0,Y 545.078,Z 516.587,A -85,B 0,C 180,E1 -3581.195,E2 -3581.195} C_VEL
LIN {X 0,Y 545.071,Z 516.589,A -85,B 0,C 180,E1 -3583.521,E2 -3583.521} C_VEL
LIN {X 0,Y 545.088,Z 516.586,A -85,B 0,C 180,E1 -3585.82,E2 -3585.82} C_VEL
LIN {X 0,Y 545.111,Z 516.578,A -85,B 0,C 180,E1 -3588.849,E2 -3588.849} C_VEL
LIN {X 0,Y 545.127,Z 516.581,A -85,B 0,C 180,E1 -3591.847,E2 -3591.847} C_VEL
LIN {X 0,Y 545.201,Z 516.567,A -85,B 0,C 180,E1 -3594.823,E2 -3594.823} C_VEL
LIN {X 0,Y 545.189,Z 516.573,A -85,B 0,C 180,E1 -3597.784,E2 -3597.784} C_VEL
LIN {X 0,Y 545.209,Z 516.566,A -85,B 0,C 180,E1 -3600.739,E2 -3600.739} C_VEL
LIN {X 0,Y 545.17,Z 516.571,A -85,B 0,C 180,E1 -3602.956,E2 -3602.956} C_VEL
LIN {X 0,Y 545.164,Z 516.576,A -85,B 0,C 180,E1 -3605.92,E2 -3605.92} C_VEL
LIN {X 0,Y 545.115,Z 516.578,A -85,B 0,C 180,E1 -3608.9,E2 -3608.9} C_VEL
LIN {X 0,Y 545.128,Z 516.581,A -85,B 0,C 180,E1 -3611.904,E2 -3611.904} C_VEL
LIN {X 0,Y 545.078,Z 516.583,A -85,B 0,C 180,E1 -3614.944,E2 -3614.944} C_VEL
LIN {X 0,Y 545.076,Z 516.586,A -85,B 0,C 180,E1 -3618.026,E2 -3618.026} C_VEL
LIN {X 0,Y 545.092,Z 516.58,A -85,B 0,C 180,E1 -3620.372,E2 -3620.372} C_VEL
LIN {X 0,Y 545.084,Z 516.589,A -85,B 0,C 180,E1 -3623.559,E2 -3623.559} C_VEL
LIN {X 0,Y 545.082,Z 516.584,A -85,B 0,C 180,E1 -3626,E2 -3626} C_VEL
LIN {X 0,Y 545.084,Z 516.582,A -85,B 0,C 180,E1 -3628.749,E2 -3628.749} C_VEL
LIN {X 0,Y 545.073,Z 516.592,A -85,B 0,C 180,E1 -3631.683,E2 -3631.683} C_VEL
LIN {X 0,Y 545.08,Z 516.581,A -85,B 0,C 180,E1 -3634.563,E2 -3634.563} C_VEL
LIN {X 0,Y 545.034,Z 516.587,A -85,B 0,C 180,E1 -3637.304,E2 -3637.304} C_VEL
LIN {X 0,Y 545.07,Z 516.586,A -85,B 0,C 180,E1 -3640.142,E2 -3640.142} C_VEL
LIN {X 0,Y 545.074,Z 516.581,A -85,B 0,C 180,E1 -3643.107,E2 -3643.107} C_VEL
LIN {X 0,Y 545.063,Z 516.585,A -85,B 0,C 180,E1 -3646.225,E2 -3646.225} C_VEL
LIN {X 0,Y 545.098,Z 516.581,A -85,B 0,C 180,E1 -3648.888,E2 -3648.888} C_VEL
LIN {X 0,Y 545.052,Z 516.587,A -85,B 0,C 180,E1 -3651.764,E2 -3651.764} C_VEL
LIN {X 0,Y 545.051,Z 516.587,A -85,B 0,C 180,E1 -3654.534,E2 -3654.534} C_VEL
LIN {X 0,Y 545.08,Z 516.581,A -85,B 0,C 180,E1 -3657.213,E2 -3657.213} C_VEL
LIN {X 0,Y 545.065,Z 516.577,A -85,B 0,C 180,E1 -3659.812,E2 -3659.812} C_VEL
LIN {X 0,Y 545.093,Z 516.581,A -85,B 0,C 180,E1 -3662.345,E2 -3662.345} C_VEL
LIN {X 0,Y 545.117,Z 516.579,A -85,B 0,C 180,E1 -3664.821,E2 -3664.821} C_VEL
LIN {X 0,Y 545.131,Z 516.812,A -85,B 0,C 180,E1 -3666.308,E2 -3666.308} C_VEL
LIN {X 0,Y 546.295,Z 523.853,A -85,B 0,C 180,E1 -3667.472,E2 -3667.472} C_VEL
LIN {X 0,Y 545.9,Z 543.109,A -85,B 0,C 180,E1 -3670.445,E2 -3670.445} C_VEL
LIN {X 0,Y 545.579,Z 560.843,A -85,B 0,C 180,E1 -3673.153,E2 -3673.153} C_VEL
LIN {X 0,Y 545.405,Z 575.941,A -85,B 0,C 180,E1 -3675.417,E2 -3675.417} C_VEL
LIN {X 0,Y 546.332,Z 582.181,A -85,B 0,C 180,E1 -3675.553,E2 -3675.553} C_VEL
LIN {X 0,Y 546.523,Z 593.984,A -85,B 0,C 180,E1 -3675.715,E2 -3675.715} C_VEL
LIN {X 0,Y 546.239,Z 683.982,A -85,B 0,C 180,E1 -3676.918,E2 -3676.918} C_VEL
LIN {X 0,Y 546.076,Z 697.234,A -85,B 0,C 180,E1 -3677.245,E2 -3677.245} C_VEL
LIN {X 0,Y 545.898,Z 710.499,A -85,B 0,C 180,E1 -3677.736,E2 -3677.736} C_VEL
LIN {X 0,Y 545.726,Z 722.38,A -85,B 0,C 180,E1 -3678.342,E2 -3678.342} C_VEL
LIN {X 0,Y 545.521,Z 733.207,A -85,B 0,C 180,E1 -3679.046,E2 -3679.046} C_VEL
LIN {X 0,Y 545.258,Z 743.612,A -85,B 0,C 180,E1 -3679.886,E2 -3679.886} C_VEL
LIN {X 0,Y 545.084,Z 752.12,A -85,B 0,C 180,E1 -3680.726,E2 -3680.726} C_VEL
LIN {X 0,Y 544.977,Z 759.966,A -85,B 0,C 180,E1 -3681.659,E2 -3681.659} C_VEL
LIN {X 0,Y 544.823,Z 767.626,A -85,B 0,C 180,E1 -3682.775,E2 -3682.775} C_VEL
LIN {X 0,Y 544.776,Z 774.682,A -85,B 0,C 180,E1 -3684.077,E2 -3684.077} C_VEL
LIN {X 0,Y 544.629,Z 779.375,A -85,B 0,C 180,E1 -3685.189,E2 -3685.189} C_VEL
LIN {X 0,Y 544.669,Z 782.962,A -85,B 0,C 180,E1 -3686.302,E2 -3686.302} C_VEL
LIN {X 0,Y 544.65,Z 784.811,A -85,B 0,C 180,E1 -3687.042,E2 -3687.042} C_VEL
LIN {X 0,Y 544.546,Z 787.185,A -85,B 0,C 180,E1 -3688.522,E2 -3688.522} C_VEL
LIN {X 0,Y 544.541,Z 788,A -85,B 0,C 180,E1 -3690.001,E2 -3690.001} C_VEL
LIN {X 0,Y 544.546,Z 787.183,A -85,B 0,C 180,E1 -3691.48,E2 -3691.48} C_VEL
LIN {X 0,Y 544.651,Z 784.806,A -85,B 0,C 180,E1 -3692.959,E2 -3692.959} C_VEL
LIN {X 0,Y 544.684,Z 781.893,A -85,B 0,C 180,E1 -3694.07,E2 -3694.07} C_VEL
LIN {X 0,Y 544.654,Z 777.947,A -85,B 0,C 180,E1 -3695.183,E2 -3695.183} C_VEL
LIN {X 0,Y 544.74,Z 772.703,A -85,B 0,C 180,E1 -3696.328,E2 -3696.328} C_VEL
LIN {X 0,Y 544.837,Z 766.463,A -85,B 0,C 180,E1 -3697.412,E2 -3697.412} C_VEL
LIN {X 0,Y 545.007,Z 758.473,A -85,B 0,C 180,E1 -3698.529,E2 -3698.529} C_VEL
LIN {X 0,Y 545.153,Z 750.328,A -85,B 0,C 180,E1 -3699.461,E2 -3699.461} C_VEL
LIN {X 0,Y 545.34,Z 740.392,A -85,B 0,C 180,E1 -3700.395,E2 -3700.395} C_VEL
LIN {X 0,Y 545.568,Z 729.583,A -85,B 0,C 180,E1 -3701.208,E2 -3701.208} C_VEL
LIN {X 0,Y 545.743,Z 718.162,A -85,B 0,C 180,E1 -3701.891,E2 -3701.891} C_VEL
LIN {X 0,Y 545.95,Z 705.968,A -85,B 0,C 180,E1 -3702.453,E2 -3702.453} C_VEL
LIN {X 0,Y 546.137,Z 693.16,A -85,B 0,C 180,E1 -3702.873,E2 -3702.873} C_VEL
LIN {X 0,Y 546.256,Z 679.563,A -85,B 0,C 180,E1 -3703.154,E2 -3703.154} C_VEL
LIN {X 0,Y 546.439,Z 582.884,A -85,B 0,C 180,E1 -3704.435,E2 -3704.435} C_VEL
LIN {X 0,Y 545.416,Z 575.983,A -85,B 0,C 180,E1 -3704.58,E2 -3704.58} C_VEL
LIN {X 0,Y 545.681,Z 555.771,A -85,B 0,C 180,E1 -3707.622,E2 -3707.622} C_VEL
LIN {X 0,Y 546.062,Z 535.458,A -85,B 0,C 180,E1 -3710.729,E2 -3710.729} C_VEL
LIN {X 0,Y 546.239,Z 522.716,A -85,B 0,C 180,E1 -3712.705,E2 -3712.705} C_VEL
LIN {X 0,Y 545.1,Z 516.712,A -85,B 0,C 180,E1 -3713.736,E2 -3713.736} C_VEL
LIN {X 0,Y 545.083,Z 516.583,A -85,B 0,C 180,E1 -3716.001,E2 -3716.001} C_VEL
LIN {X 0,Y 545.079,Z 516.575,A -85,B 0,C 180,E1 -3718.746,E2 -3718.746} C_VEL
LIN {X 0,Y 545.062,Z 516.589,A -85,B 0,C 180,E1 -3721.679,E2 -3721.679} C_VEL
LIN {X 0,Y 545.066,Z 516.587,A -85,B 0,C 180,E1 -3724.565,E2 -3724.565} C_VEL
LIN {X 0,Y 545.04,Z 516.588,A -85,B 0,C 180,E1 -3727.304,E2 -3727.304} C_VEL
LIN {X 0,Y 545.071,Z 516.591,A -85,B 0,C 180,E1 -3730.143,E2 -3730.143} C_VEL
LIN {X 0,Y 545.086,Z 516.582,A -85,B 0,C 180,E1 -3733.106,E2 -3733.106} C_VEL
LIN {X 0,Y 545.071,Z 516.59,A -85,B 0,C 180,E1 -3736.224,E2 -3736.224} C_VEL
LIN {X 0,Y 545.101,Z 516.581,A -85,B 0,C 180,E1 -3738.887,E2 -3738.887} C_VEL
LIN {X 0,Y 545.058,Z 516.593,A -85,B 0,C 180,E1 -3741.763,E2 -3741.763} C_VEL
LIN {X 0,Y 545.069,Z 516.586,A -85,B 0,C 180,E1 -3744.534,E2 -3744.534} C_VEL
LIN {X 0,Y 545.085,Z 516.585,A -85,B 0,C 180,E1 -3747.213,E2 -3747.213} C_VEL
LIN {X 0,Y 545.068,Z 516.594,A -85,B 0,C 180,E1 -3749.811,E2 -3749.811} C_VEL
LIN {X 0,Y 545.084,Z 516.587,A -85,B 0,C 180,E1 -3752.344,E2 -3752.344} C_VEL
LIN {X 0,Y 545.164,Z 516.793,A -85,B 0,C 180,E1 -3754.363,E2 -3754.363} C_VEL
LIN {X 0,Y 546.422,Z 523.741,A -85,B 0,C 180,E1 -3755.291,E2 -3755.291} C_VEL
LIN {X 0,Y 546.351,Z 540.436,A -85,B 0,C 180,E1 -3757.465,E2 -3757.465} C_VEL
LIN {X 0,Y 546.169,Z 555.942,A -85,B 0,C 180,E1 -3759.473,E2 -3759.473} C_VEL
LIN {X 0,Y 545.861,Z 577.438,A -85,B 0,C 180,E1 -3762.318,E2 -3762.318} C_VEL
LIN {X 0,Y 545.495,Z 598.959,A -85,B 0,C 180,E1 -3765.218,E2 -3765.218} C_VEL
LIN {X 0,Y 545.194,Z 621.581,A -85,B 0,C 180,E1 -3768.231,E2 -3768.231} C_VEL
LIN {X 0,Y 545.141,Z 631.029,A -85,B 0,C 180,E1 -3769.461,E2 -3769.461} C_VEL
LIN {X 0,Y 545.639,Z 637.949,A -85,B 0,C 180,E1 -3769.588,E2 -3769.588} C_VEL
LIN {X 0,Y 545.48,Z 702.473,A -85,B 0,C 180,E1 -3770.452,E2 -3770.452} C_VEL
LIN {X 0,Y 545.395,Z 714.467,A -85,B 0,C 180,E1 -3770.777,E2 -3770.777} C_VEL
LIN {X 0,Y 545.313,Z 724.458,A -85,B 0,C 180,E1 -3771.197,E2 -3771.197} C_VEL
LIN {X 0,Y 545.171,Z 734.238,A -85,B 0,C 180,E1 -3771.754,E2 -3771.754} C_VEL
LIN {X 0,Y 545,Z 744.049,A -85,B 0,C 180,E1 -3772.498,E2 -3772.498} C_VEL
LIN {X 0,Y 544.887,Z 752.549,A -85,B 0,C 180,E1 -3773.334,E2 -3773.334} C_VEL
LIN {X 0,Y 544.819,Z 759.94,A -85,B 0,C 180,E1 -3774.262,E2 -3774.262} C_VEL
LIN {X 0,Y 544.773,Z 765.682,A -85,B 0,C 180,E1 -3775.19,E2 -3775.19} C_VEL
LIN {X 0,Y 544.692,Z 770.864,A -85,B 0,C 180,E1 -3776.301,E2 -3776.301} C_VEL
LIN {X 0,Y 544.669,Z 773.465,A -85,B 0,C 180,E1 -3777.042,E2 -3777.042} C_VEL
LIN {X 0,Y 544.57,Z 775.421,A -85,B 0,C 180,E1 -3777.781,E2 -3777.781} C_VEL
LIN {X 0,Y 544.542,Z 776.829,A -85,B 0,C 180,E1 -3778.521,E2 -3778.521} C_VEL
LIN {X 0,Y 544.537,Z 777.683,A -85,B 0,C 180,E1 -3779.261,E2 -3779.261} C_VEL
LIN {X 0,Y 544.539,Z 777.996,A -85,B 0,C 180,E1 -3780,E2 -3780} C_VEL
LIN {X 0,Y 544.539,Z 777.759,A -85,B 0,C 180,E1 -3780.74,E2 -3780.74} C_VEL
LIN {X 0,Y 544.545,Z 776.968,A -85,B 0,C 180,E1 -3781.479,E2 -3781.479} C_VEL
LIN {X 0,Y 544.569,Z 775.618,A -85,B 0,C 180,E1 -3782.219,E2 -3782.219} C_VEL
LIN {X 0,Y 544.691,Z 772.556,A -85,B 0,C 180,E1 -3783.329,E2 -3783.329} C_VEL
LIN {X 0,Y 544.729,Z 768.019,A -85,B 0,C 180,E1 -3784.44,E2 -3784.44} C_VEL
LIN {X 0,Y 544.716,Z 762.956,A -85,B 0,C 180,E1 -3785.367,E2 -3785.367} C_VEL
LIN {X 0,Y 544.917,Z 756.998,A -85,B 0,C 180,E1 -3786.225,E2 -3786.225} C_VEL
LIN {X 0,Y 544.926,Z 749.955,A -85,B 0,C 180,E1 -3787.037,E2 -3787.037} C_VEL
LIN {X 0,Y 545.075,Z 740.617,A -85,B 0,C 180,E1 -3787.874,E2 -3787.874} C_VEL
LIN {X 0,Y 545.229,Z 731.185,A -85,B 0,C 180,E1 -3788.525,E2 -3788.525} C_VEL
LIN {X 0,Y 545.386,Z 720.371,A -85,B 0,C 180,E1 -3789.083,E2 -3789.083} C_VEL
LIN {X 0,Y 545.439,Z 709.125,A -85,B 0,C 180,E1 -3789.479,E2 -3789.479} C_VEL
LIN {X 0,Y 545.494,Z 698.262,A -85,B 0,C 180,E1 -3789.712,E2 -3789.712} C_VEL
LIN {X 0,Y 545.604,Z 635.864,A -85,B 0,C 180,E1 -3790.53,E2 -3790.53} C_VEL
LIN {X 0,Y 545.107,Z 630.972,A -85,B 0,C 180,E1 -3790.634,E2 -3790.634} C_VEL
LIN {X 0,Y 545.375,Z 607.04,A -85,B 0,C 180,E1 -3793.792,E2 -3793.792} C_VEL
LIN {X 0,Y 545.712,Z 585.721,A -85,B 0,C 180,E1 -3796.652,E2 -3796.652} C_VEL
LIN {X 0,Y 546.045,Z 565.546,A -85,B 0,C 180,E1 -3799.355,E2 -3799.355} C_VEL
LIN {X 0,Y 546.431,Z 541.85,A -85,B 0,C 180,E1 -3802.536,E2 -3802.536} C_VEL
LIN {X 0,Y 546.671,Z 527.559,A -85,B 0,C 180,E1 -3804.468,E2 -3804.468} C_VEL
LIN {X 0,Y 546.047,Z 525.82,A -85,B 0,C 180,E1 -3804.734,E2 -3804.734} C_VEL
LIN {X 0,Y 543.89,Z 523.821,A -85,B 0,C 180,E1 -3805.093,E2 -3805.093} C_VEL
LIN {X 0,Y 538.947,Z 519.604,A -85,B 0,C 180,E1 -3805.827,E2 -3805.827} C_VEL
LIN {X 0,Y 538.091,Z 517.568,A -85,B 0,C 180,E1 -3806.193,E2 -3806.193} C_VEL
LIN {X 0,Y 538.077,Z 517.519,A -85,B 0,C 180,E1 -3806.232,E2 -3806.232} C_VEL
LIN {X 0,Y 538.035,Z 517.465,A -85,B 0,C 180,E1 -3808.933,E2 -3808.933} C_VEL
LIN {X 0,Y 538.015,Z 517.466,A -85,B 0,C 180,E1 -3811.887,E2 -3811.887} C_VEL
LIN {X 0,Y 538.036,Z 517.467,A -85,B 0,C 180,E1 -3814.621,E2 -3814.621} C_VEL
LIN {X 0,Y 538.015,Z 517.463,A -85,B 0,C 180,E1 -3817.171,E2 -3817.171} C_VEL
LIN {X 0,Y 538.031,Z 517.46,A -85,B 0,C 180,E1 -3819.797,E2 -3819.797} C_VEL
LIN {X 0,Y 538.023,Z 517.458,A -85,B 0,C 180,E1 -3822.786,E2 -3822.786} C_VEL
LIN {X 0,Y 538.034,Z 517.46,A -85,B 0,C 180,E1 -3825.925,E2 -3825.925} C_VEL
LIN {X 0,Y 538.054,Z 517.454,A -85,B 0,C 180,E1 -3829.224,E2 -3829.224} C_VEL
LIN {X 0,Y 537.997,Z 517.464,A -85,B 0,C 180,E1 -3832.122,E2 -3832.122} C_VEL
LIN {X 0,Y 538.003,Z 517.466,A -85,B 0,C 180,E1 -3834.915,E2 -3834.915} C_VEL
LIN {X 0,Y 538.024,Z 517.461,A -85,B 0,C 180,E1 -3837.617,E2 -3837.617} C_VEL
LIN {X 0,Y 538.022,Z 517.466,A -85,B 0,C 180,E1 -3840.239,E2 -3840.239} C_VEL
LIN {X 0,Y 538.062,Z 517.464,A -85,B 0,C 180,E1 -3842.796,E2 -3842.796} C_VEL
LIN {X 0,Y 538.033,Z 517.459,A -85,B 0,C 180,E1 -3845.291,E2 -3845.291} C_VEL
LIN {X 0,Y 538.021,Z 517.464,A -85,B 0,C 180,E1 -3848.042,E2 -3848.042} C_VEL
LIN {X 0,Y 538.116,Z 517.638,A -85,B 0,C 180,E1 -3849.693,E2 -3849.693} C_VEL
LIN {X 0,Y 538.671,Z 523.032,A -85,B 0,C 180,E1 -3850.765,E2 -3850.765} C_VEL
LIN {X 0,Y 538.349,Z 538.596,A -85,B 0,C 180,E1 -3853.699,E2 -3853.699} C_VEL
LIN {X 0,Y 538.25,Z 544.993,A -85,B 0,C 180,E1 -3854.862,E2 -3854.862} C_VEL
LIN {X 0,Y 538.304,Z 548.254,A -85,B 0,C 180,E1 -3855.301,E2 -3855.301} C_VEL
LIN {X 0,Y 539.681,Z 556.839,A -85,B 0,C 180,E1 -3855.478,E2 -3855.478} C_VEL
LIN {X 0,Y 539.328,Z 654.058,A -85,B 0,C 180,E1 -3856.794,E2 -3856.794} C_VEL
LIN {X 0,Y 539.164,Z 667.294,A -85,B 0,C 180,E1 -3857.125,E2 -3857.125} C_VEL
LIN {X 0,Y 538.951,Z 679.427,A -85,B 0,C 180,E1 -3857.574,E2 -3857.574} C_VEL
LIN {X 0,Y 538.746,Z 691.615,A -85,B 0,C 180,E1 -3858.188,E2 -3858.188} C_VEL
LIN {X 0,Y 538.548,Z 702.577,A -85,B 0,C 180,E1 -3858.901,E2 -3858.901} C_VEL
LIN {X 0,Y 538.278,Z 713.092,A -85,B 0,C 180,E1 -3859.752,E2 -3859.752} C_VEL
LIN {X 0,Y 538.086,Z 721.688,A -85,B 0,C 180,E1 -3860.603,E2 -3860.603} C_VEL
LIN {X 0,Y 537.923,Z 729.605,A -85,B 0,C 180,E1 -3861.547,E2 -3861.547} C_VEL
LIN {X 0,Y 537.759,Z 737.351,A -85,B 0,C 180,E1 -3862.679,E2 -3862.679} C_VEL
LIN {X 0,Y 537.694,Z 744.461,A -85,B 0,C 180,E1 -3863.997,E2 -3863.997} C_VEL
LIN {X 0,Y 537.54,Z 749.201,A -85,B 0,C 180,E1 -3865.124,E2 -3865.124} C_VEL
LIN {X 0,Y 537.591,Z 752.831,A -85,B 0,C 180,E1 -3866.252,E2 -3866.252} C_VEL
LIN {X 0,Y 537.551,Z 754.709,A -85,B 0,C 180,E1 -3867.002,E2 -3867.002} C_VEL
LIN {X 0,Y 537.49,Z 756.129,A -85,B 0,C 180,E1 -3867.751,E2 -3867.751} C_VEL
LIN {X 0,Y 537.442,Z 757.757,A -85,B 0,C 180,E1 -3869.25,E2 -3869.25} C_VEL
LIN {X 0,Y 537.442,Z 757.996,A -85,B 0,C 180,E1 -3869.999,E2 -3869.999} C_VEL
LIN {X 0,Y 537.442,Z 757.814,A -85,B 0,C 180,E1 -3870.749,E2 -3870.749} C_VEL
LIN {X 0,Y 537.49,Z 756.266,A -85,B 0,C 180,E1 -3872.247,E2 -3872.247} C_VEL
LIN {X 0,Y 537.552,Z 754.905,A -85,B 0,C 180,E1 -3872.997,E2 -3872.997} C_VEL
LIN {X 0,Y 537.604,Z 752.024,A -85,B 0,C 180,E1 -3874.122,E2 -3874.122} C_VEL
LIN {X 0,Y 537.587,Z 748.122,A -85,B 0,C 180,E1 -3875.25,E2 -3875.25} C_VEL
LIN {X 0,Y 537.638,Z 743.37,A -85,B 0,C 180,E1 -3876.32,E2 -3876.32} C_VEL
LIN {X 0,Y 537.789,Z 736.762,A -85,B 0,C 180,E1 -3877.508,E2 -3877.508} C_VEL
LIN {X 0,Y 537.969,Z 728.836,A -85,B 0,C 180,E1 -3878.64,E2 -3878.64} C_VEL
LIN {X 0,Y 538.112,Z 720.763,A -85,B 0,C 180,E1 -3879.585,E2 -3879.585} C_VEL
LIN {X 0,Y 538.347,Z 710.911,A -85,B 0,C 180,E1 -3880.53,E2 -3880.53} C_VEL
LIN {X 0,Y 538.58,Z 701.23,A -85,B 0,C 180,E1 -3881.287,E2 -3881.287} C_VEL
LIN {X 0,Y 538.742,Z 690.722,A -85,B 0,C 180,E1 -3881.954,E2 -3881.954} C_VEL
LIN {X 0,Y 538.988,Z 678.193,A -85,B 0,C 180,E1 -3882.567,E2 -3882.567} C_VEL
LIN {X 0,Y 539.181,Z 664.861,A -85,B 0,C 180,E1 -3883.041,E2 -3883.041} C_VEL
LIN {X 0,Y 539.362,Z 652.48,A -85,B 0,C 180,E1 -3883.324,E2 -3883.324} C_VEL
LIN {X 0,Y 539.65,Z 555.829,A -85,B 0,C 180,E1 -3884.626,E2 -3884.626} C_VEL
LIN {X 0,Y 538.369,Z 548.53,A -85,B 0,C 180,E1 -3884.77,E2 -3884.77} C_VEL
LIN {X 0,Y 538.267,Z 545.599,A -85,B 0,C 180,E1 -3885.137,E2 -3885.137} C_VEL
LIN {X 0,Y 538.441,Z 532.885,A -85,B 0,C 180,E1 -3887.469,E2 -3887.469} C_VEL
LIN {X 0,Y 538.624,Z 521.449,A -85,B 0,C 180,E1 -3889.632,E2 -3889.632} C_VEL
LIN {X 0,Y 538.064,Z 517.51,A -85,B 0,C 180,E1 -3890.458,E2 -3890.458} C_VEL
LIN {X 0,Y 538.024,Z 517.469,A -85,B 0,C 180,E1 -3893.071,E2 -3893.071} C_VEL
LIN {X 0,Y 538.044,Z 517.462,A -85,B 0,C 180,E1 -3895.672,E2 -3895.672} C_VEL
LIN {X 0,Y 538.045,Z 517.46,A -85,B 0,C 180,E1 -3898.049,E2 -3898.049} C_VEL
LIN {X 0,Y 538.02,Z 517.461,A -85,B 0,C 180,E1 -3900.626,E2 -3900.626} C_VEL
LIN {X 0,Y 538.044,Z 517.466,A -85,B 0,C 180,E1 -3903.282,E2 -3903.282} C_VEL
LIN {X 0,Y 538.026,Z 517.461,A -85,B 0,C 180,E1 -3906.001,E2 -3906.001} C_VEL
LIN {X 0,Y 538.014,Z 517.464,A -85,B 0,C 180,E1 -3908.829,E2 -3908.829} C_VEL
LIN {X 0,Y 538.035,Z 517.463,A -85,B 0,C 180,E1 -3911.879,E2 -3911.879} C_VEL
LIN {X 0,Y 538.028,Z 517.462,A -85,B 0,C 180,E1 -3915.14,E2 -3915.14} C_VEL
LIN {X 0,Y 538.037,Z 517.46,A -85,B 0,C 180,E1 -3918.227,E2 -3918.227} C_VEL
LIN {X 0,Y 538.055,Z 517.454,A -85,B 0,C 180,E1 -3920.411,E2 -3920.411} C_VEL
LIN {X 0,Y 538.028,Z 517.461,A -85,B 0,C 180,E1 -3923.067,E2 -3923.067} C_VEL
LIN {X 0,Y 538.028,Z 517.464,A -85,B 0,C 180,E1 -3925.827,E2 -3925.827} C_VEL
LIN {X 0,Y 538.019,Z 517.461,A -85,B 0,C 180,E1 -3928.499,E2 -3928.499} C_VEL
LIN {X 0,Y 538.053,Z 517.461,A -85,B 0,C 180,E1 -3931.099,E2 -3931.099} C_VEL
LIN {X 0,Y 538.045,Z 517.466,A -85,B 0,C 180,E1 -3933.633,E2 -3933.633} C_VEL
LIN {X 0,Y 538.016,Z 517.462,A -85,B 0,C 180,E1 -3936.117,E2 -3936.117} C_VEL
LIN {X 0,Y 538.036,Z 517.465,A -85,B 0,C 180,E1 -3939.348,E2 -3939.348} C_VEL
LIN {X 0,Y 538.066,Z 517.454,A -85,B 0,C 180,E1 -3942.517,E2 -3942.517} C_VEL
LIN {X 0,Y 538.057,Z 517.465,A -85,B 0,C 180,E1 -3945.63,E2 -3945.63} C_VEL
LIN {X 0,Y 538.07,Z 517.454,A -85,B 0,C 180,E1 -3948.701,E2 -3948.701} C_VEL
LIN {X 0,Y 538.083,Z 517.46,A -85,B 0,C 180,E1 -3951.739,E2 -3951.739} C_VEL
LIN {X 0,Y 538.158,Z 517.444,A -85,B 0,C 180,E1 -3954.755,E2 -3954.755} C_VEL
LIN {X 0,Y 538.161,Z 517.449,A -85,B 0,C 180,E1 -3957.755,E2 -3957.755} C_VEL
LIN {X 0,Y 538.178,Z 517.442,A -85,B 0,C 180,E1 -3960.748,E2 -3960.748} C_VEL
LIN {X 0,Y 538.136,Z 517.447,A -85,B 0,C 180,E1 -3962.994,E2 -3962.994} C_VEL
LIN {X 0,Y 538.117,Z 517.453,A -85,B 0,C 180,E1 -3965.997,E2 -3965.997} C_VEL
LIN {X 0,Y 538.065,Z 517.457,A -85,B 0,C 180,E1 -3969.018,E2 -3969.018} C_VEL
LIN {X 0,Y 538.076,Z 517.457,A -85,B 0,C 180,E1 -3972.063,E2 -3972.063} C_VEL
LIN {X 0,Y 538.038,Z 517.461,A -85,B 0,C 180,E1 -3975.144,E2 -3975.144} C_VEL
LIN {X 0,Y 538.028,Z 517.461,A -85,B 0,C 180,E1 -3978.27,E2 -3978.27} C_VEL
LIN {X 0,Y 538.036,Z 517.459,A -85,B 0,C 180,E1 -3980.652,E2 -3980.652} C_VEL
LIN {X 0,Y 538.017,Z 517.467,A -85,B 0,C 180,E1 -3983.888,E2 -3983.888} C_VEL
LIN {X 0,Y 538.044,Z 517.457,A -85,B 0,C 180,E1 -3986.367,E2 -3986.367} C_VEL
LIN {X 0,Y 538.025,Z 517.462,A -85,B 0,C 180,E1 -3988.934,E2 -3988.934} C_VEL
LIN {X 0,Y 538.022,Z 517.467,A -85,B 0,C 180,E1 -3991.891,E2 -3991.891} C_VEL
LIN {X 0,Y 538.029,Z 517.459,A -85,B 0,C 180,E1 -3994.622,E2 -3994.622} C_VEL
LIN {X 0,Y 538.002,Z 517.461,A -85,B 0,C 180,E1 -3997.171,E2 -3997.171} C_VEL
LIN {X 0,Y 538.025,Z 517.468,A -85,B 0,C 180,E1 -3999.797,E2 -3999.797} C_VEL
LIN {X 0,Y 538.015,Z 517.459,A -85,B 0,C 180,E1 -4002.787,E2 -4002.787} C_VEL
LIN {X 0,Y 538.026,Z 517.465,A -85,B 0,C 180,E1 -4005.926,E2 -4005.926} C_VEL
LIN {X 0,Y 538.075,Z 517.458,A -85,B 0,C 180,E1 -4009.25,E2 -4009.25} C_VEL
LIN {X 0,Y 537.991,Z 517.464,A -85,B 0,C 180,E1 -4012.123,E2 -4012.123} C_VEL
LIN {X 0,Y 538.01,Z 517.464,A -85,B 0,C 180,E1 -4014.918,E2 -4014.918} C_VEL
LIN {X 0,Y 538.03,Z 517.454,A -85,B 0,C 180,E1 -4017.619,E2 -4017.619} C_VEL
LIN {X 0,Y 538.017,Z 517.464,A -85,B 0,C 180,E1 -4020.24,E2 -4020.24} C_VEL
LIN {X 0,Y 538.066,Z 517.455,A -85,B 0,C 180,E1 -4022.797,E2 -4022.797} C_VEL
LIN {X 0,Y 538.031,Z 517.468,A -85,B 0,C 180,E1 -4025.704,E2 -4025.704} C_VEL
LIN {X 0,Y 538.101,Z 517.732,A -85,B 0,C 180,E1 -4026.158,E2 -4026.158} C_VEL
LIN {X 0,Y 539.343,Z 525.378,A -85,B 0,C 180,E1 -4027.435,E2 -4027.435} C_VEL
LIN {X 0,Y 538.924,Z 544.203,A -85,B 0,C 180,E1 -4030.38,E2 -4030.38} C_VEL
LIN {X 0,Y 538.56,Z 562.012,A -85,B 0,C 180,E1 -4033.122,E2 -4033.122} C_VEL
LIN {X 0,Y 538.39,Z 575.944,A -85,B 0,C 180,E1 -4035.222,E2 -4035.222} C_VEL
LIN {X 0,Y 539.233,Z 581.432,A -85,B 0,C 180,E1 -4035.348,E2 -4035.348} C_VEL
LIN {X 0,Y 539.698,Z 587.31,A -85,B 0,C 180,E1 -4035.44,E2 -4035.44} C_VEL
LIN {X 0,Y 539.34,Z 683.982,A -85,B 0,C 180,E1 -4036.747,E2 -4036.747} C_VEL
LIN {X 0,Y 539.149,Z 697.232,A -85,B 0,C 180,E1 -4037.078,E2 -4037.078} C_VEL
LIN {X 0,Y 538.951,Z 710.499,A -85,B 0,C 180,E1 -4037.576,E2 -4037.576} C_VEL
LIN {X 0,Y 538.744,Z 722.379,A -85,B 0,C 180,E1 -4038.189,E2 -4038.189} C_VEL
LIN {X 0,Y 538.515,Z 734.496,A -85,B 0,C 180,E1 -4038.997,E2 -4038.997} C_VEL
LIN {X 0,Y 538.228,Z 744.653,A -85,B 0,C 180,E1 -4039.848,E2 -4039.848} C_VEL
LIN {X 0,Y 538.026,Z 753.792,A -85,B 0,C 180,E1 -4040.793,E2 -4040.793} C_VEL
LIN {X 0,Y 537.85,Z 762.693,A -85,B 0,C 180,E1 -4041.926,E2 -4041.926} C_VEL
LIN {X 0,Y 537.728,Z 769.853,A -85,B 0,C 180,E1 -4043.057,E2 -4043.057} C_VEL
LIN {X 0,Y 537.676,Z 776.368,A -85,B 0,C 180,E1 -4044.375,E2 -4044.375} C_VEL
LIN {X 0,Y 537.557,Z 780.679,A -85,B 0,C 180,E1 -4045.502,E2 -4045.502} C_VEL
LIN {X 0,Y 537.591,Z 782.963,A -85,B 0,C 180,E1 -4046.253,E2 -4046.253} C_VEL
LIN {X 0,Y 537.551,Z 784.811,A -85,B 0,C 180,E1 -4047.003,E2 -4047.003} C_VEL
LIN {X 0,Y 537.451,Z 787.185,A -85,B 0,C 180,E1 -4048.502,E2 -4048.502} C_VEL
LIN {X 0,Y 537.442,Z 788,A -85,B 0,C 180,E1 -4050.001,E2 -4050.001} C_VEL
LIN {X 0,Y 537.451,Z 787.182,A -85,B 0,C 180,E1 -4051.499,E2 -4051.499} C_VEL
LIN {X 0,Y 537.551,Z 784.806,A -85,B 0,C 180,E1 -4052.998,E2 -4052.998} C_VEL
LIN {X 0,Y 537.603,Z 781.893,A -85,B 0,C 180,E1 -4054.124,E2 -4054.124} C_VEL
LIN {X 0,Y 537.588,Z 777.947,A -85,B 0,C 180,E1 -4055.251,E2 -4055.251} C_VEL
LIN {X 0,Y 537.651,Z 773.08,A -85,B 0,C 180,E1 -4056.335,E2 -4056.335} C_VEL
LIN {X 0,Y 537.791,Z 766.462,A -85,B 0,C 180,E1 -4057.51,E2 -4057.51} C_VEL
LIN {X 0,Y 537.973,Z 758.473,A -85,B 0,C 180,E1 -4058.641,E2 -4058.641} C_VEL
LIN {X 0,Y 538.144,Z 750.327,A -85,B 0,C 180,E1 -4059.586,E2 -4059.586} C_VEL
LIN {X 0,Y 538.34,Z 740.392,A -85,B 0,C 180,E1 -4060.532,E2 -4060.532} C_VEL
LIN {X 0,Y 538.577,Z 730.58,A -85,B 0,C 180,E1 -4061.288,E2 -4061.288} C_VEL
LIN {X 0,Y 538.754,Z 719.532,A -85,B 0,C 180,E1 -4061.974,E2 -4061.974} C_VEL
LIN {X 0,Y 539.002,Z 707.096,A -85,B 0,C 180,E1 -4062.568,E2 -4062.568} C_VEL
LIN {X 0,Y 539.222,Z 694.073,A -85,B 0,C 180,E1 -4063.017,E2 -4063.017} C_VEL
LIN {X 0,Y 539.377,Z 681.067,A -85,B 0,C 180,E1 -4063.301,E2 -4063.301} C_VEL
LIN {X 0,Y 539.57,Z 583.665,A -85,B 0,C 180,E1 -4064.612,E2 -4064.612} C_VEL
LIN {X 0,Y 538.384,Z 576.043,A -85,B 0,C 180,E1 -4064.771,E2 -4064.771} C_VEL
LIN {X 0,Y 538.693,Z 556.313,A -85,B 0,C 180,E1 -4067.751,E2 -4067.751} C_VEL
LIN {X 0,Y 539.091,Z 536.56,A -85,B 0,C 180,E1 -4070.809,E2 -4070.809} C_VEL
LIN {X 0,Y 539.263,Z 523.829,A -85,B 0,C 180,E1 -4072.813,E2 -4072.813} C_VEL
LIN {X 0,Y 538.038,Z 517.552,A -85,B 0,C 180,E1 -4073.913,E2 -4073.913} C_VEL
LIN {X 0,Y 538.046,Z 517.463,A -85,B 0,C 180,E1 -4076.367,E2 -4076.367} C_VEL
LIN {X 0,Y 538.034,Z 517.45,A -85,B 0,C 180,E1 -4078.934,E2 -4078.934} C_VEL
LIN {X 0,Y 538.014,Z 517.469,A -85,B 0,C 180,E1 -4081.887,E2 -4081.887} C_VEL
LIN {X 0,Y 538.016,Z 517.465,A -85,B 0,C 180,E1 -4084.618,E2 -4084.618} C_VEL
LIN {X 0,Y 538.008,Z 517.463,A -85,B 0,C 180,E1 -4087.17,E2 -4087.17} C_VEL
LIN {X 0,Y 538.028,Z 517.467,A -85,B 0,C 180,E1 -4089.797,E2 -4089.797} C_VEL
LIN {X 0,Y 538.025,Z 517.462,A -85,B 0,C 180,E1 -4092.786,E2 -4092.786} C_VEL
LIN {X 0,Y 538.034,Z 517.468,A -85,B 0,C 180,E1 -4095.926,E2 -4095.926} C_VEL
LIN {X 0,Y 538.056,Z 517.46,A -85,B 0,C 180,E1 -4099.252,E2 -4099.252} C_VEL
LIN {X 0,Y 537.998,Z 517.472,A -85,B 0,C 180,E1 -4102.123,E2 -4102.123} C_VEL
LIN {X 0,Y 538.024,Z 517.462,A -85,B 0,C 180,E1 -4104.917,E2 -4104.917} C_VEL
LIN {X 0,Y 538.03,Z 517.468,A -85,B 0,C 180,E1 -4107.618,E2 -4107.618} C_VEL
LIN {X 0,Y 538.021,Z 517.467,A -85,B 0,C 180,E1 -4110.239,E2 -4110.239} C_VEL
LIN {X 0,Y 538.06,Z 517.461,A -85,B 0,C 180,E1 -4112.796,E2 -4112.796} C_VEL
LIN {X 0,Y 538.13,Z 517.687,A -85,B 0,C 180,E1 -4114.279,E2 -4114.279} C_VEL
LIN {X 0,Y 539.484,Z 525.772,A -85,B 0,C 180,E1 -4115.363,E2 -4115.363} C_VEL
LIN {X 0,Y 539.329,Z 544.583,A -85,B 0,C 180,E1 -4117.796,E2 -4117.796} C_VEL
LIN {X 0,Y 539.094,Z 560.766,A -85,B 0,C 180,E1 -4119.93,E2 -4119.93} C_VEL
LIN {X 0,Y 538.805,Z 580.589,A -85,B 0,C 180,E1 -4122.542,E2 -4122.542} C_VEL
LIN {X 0,Y 538.443,Z 603.531,A -85,B 0,C 180,E1 -4125.641,E2 -4125.641} C_VEL
LIN {X 0,Y 538.116,Z 627.683,A -85,B 0,C 180,E1 -4128.893,E2 -4128.893} C_VEL
LIN {X 0,Y 538.122,Z 631.043,A -85,B 0,C 180,E1 -4129.322,E2 -4129.322} C_VEL
LIN {X 0,Y 538.661,Z 637.995,A -85,B 0,C 180,E1 -4129.451,E2 -4129.451} C_VEL
LIN {X 0,Y 538.482,Z 702.496,A -85,B 0,C 180,E1 -4130.326,E2 -4130.326} C_VEL
LIN {X 0,Y 538.392,Z 714.478,A -85,B 0,C 180,E1 -4130.656,E2 -4130.656} C_VEL
LIN {X 0,Y 538.304,Z 724.479,A -85,B 0,C 180,E1 -4131.081,E2 -4131.081} C_VEL
LIN {X 0,Y 538.142,Z 734.253,A -85,B 0,C 180,E1 -4131.646,E2 -4131.646} C_VEL
LIN {X 0,Y 537.949,Z 744.055,A -85,B 0,C 180,E1 -4132.399,E2 -4132.399} C_VEL
LIN {X 0,Y 537.829,Z 752.831,A -85,B 0,C 180,E1 -4133.277,E2 -4133.277} C_VEL
LIN {X 0,Y 537.77,Z 759.943,A -85,B 0,C 180,E1 -4134.187,E2 -4134.187} C_VEL
LIN {X 0,Y 537.676,Z 765.687,A -85,B 0,C 180,E1 -4135.126,E2 -4135.126} C_VEL
LIN {X 0,Y 537.614,Z 770.872,A -85,B 0,C 180,E1 -4136.252,E2 -4136.252} C_VEL
LIN {X 0,Y 537.602,Z 773.473,A -85,B 0,C 180,E1 -4137.003,E2 -4137.003} C_VEL
LIN {X 0,Y 537.49,Z 775.425,A -85,B 0,C 180,E1 -4137.752,E2 -4137.752} C_VEL
LIN {X 0,Y 537.448,Z 776.827,A -85,B 0,C 180,E1 -4138.501,E2 -4138.501} C_VEL
LIN {X 0,Y 537.437,Z 777.681,A -85,B 0,C 180,E1 -4139.251,E2 -4139.251} C_VEL
LIN {X 0,Y 537.44,Z 777.996,A -85,B 0,C 180,E1 -4140,E2 -4140} C_VEL
LIN {X 0,Y 537.44,Z 777.759,A -85,B 0,C 180,E1 -4140.749,E2 -4140.749} C_VEL
LIN {X 0,Y 537.451,Z 776.965,A -85,B 0,C 180,E1 -4141.499,E2 -4141.499} C_VEL
LIN {X 0,Y 537.488,Z 775.619,A -85,B 0,C 180,E1 -4142.248,E2 -4142.248} C_VEL
LIN {X 0,Y 537.591,Z 772.552,A -85,B 0,C 180,E1 -4143.373,E2 -4143.373} C_VEL
LIN {X 0,Y 537.634,Z 768.015,A -85,B 0,C 180,E1 -4144.499,E2 -4144.499} C_VEL
LIN {X 0,Y 537.656,Z 762.958,A -85,B 0,C 180,E1 -4145.438,E2 -4145.438} C_VEL
LIN {X 0,Y 537.84,Z 757.53,A -85,B 0,C 180,E1 -4146.237,E2 -4146.237} C_VEL
LIN {X 0,Y 537.868,Z 749.945,A -85,B 0,C 180,E1 -4147.131,E2 -4147.131} C_VEL
LIN {X 0,Y 538.001,Z 741.794,A -85,B 0,C 180,E1 -4147.884,E2 -4147.884} C_VEL
LIN {X 0,Y 538.2,Z 732.692,A -85,B 0,C 180,E1 -4148.542,E2 -4148.542} C_VEL
LIN {X 0,Y 538.319,Z 722.389,A -85,B 0,C 180,E1 -4149.108,E2 -4149.108} C_VEL
LIN {X 0,Y 538.439,Z 711.531,A -85,B 0,C 180,E1 -4149.532,E2 -4149.532} C_VEL
LIN {X 0,Y 538.519,Z 701.094,A -85,B 0,C 180,E1 -4149.792,E2 -4149.792} C_VEL
LIN {X 0,Y 538.549,Z 635.818,A -85,B 0,C 180,E1 -4150.67,E2 -4150.67} C_VEL
LIN {X 0,Y 538.09,Z 630.969,A -85,B 0,C 180,E1 -4150.774,E2 -4150.774} C_VEL
LIN {X 0,Y 538.364,Z 607.035,A -85,B 0,C 180,E1 -4153.976,E2 -4153.976} C_VEL
LIN {X 0,Y 538.732,Z 585.615,A -85,B 0,C 180,E1 -4156.874,E2 -4156.874} C_VEL
LIN {X 0,Y 539.049,Z 566.631,A -85,B 0,C 180,E1 -4159.418,E2 -4159.418} C_VEL
LIN {X 0,Y 539.458,Z 545.061,A -85,B 0,C 180,E1 -4162.334,E2 -4162.334} C_VEL
LIN {X 0,Y 539.723,Z 526.711,A -85,B 0,C 180,E1 -4164.831,E2 -4164.831} C_VEL
LIN {X 0,Y 538.105,Z 517.565,A -85,B 0,C 180,E1 -4166.173,E2 -4166.173} C_VEL
LIN {X 0,Y 538.077,Z 517.519,A -85,B 0,C 180,E1 -4166.232,E2 -4166.232} C_VEL
LIN {X 0,Y 537.338,Z 517.555,A -85,B 0,C 180,E1 -4166.856,E2 -4166.856} C_VEL
LIN {X 0,Y 534.472,Z 517.911,A -85,B 0,C 180,E1 -4167.87,E2 -4167.87} C_VEL
LIN {X 0,Y 532.089,Z 518.223,A -85,B 0,C 180,E1 -4168.687,E2 -4168.687} C_VEL
LIN {X 0,Y 531.061,Z 518.333,A -85,B 0,C 180,E1 -4169.318,E2 -4169.318} C_VEL
LIN {X 0,Y 530.972,Z 518.342,A -85,B 0,C 180,E1 -4169.531,E2 -4169.531} C_VEL
LIN {X 0,Y 530.97,Z 518.346,A -85,B 0,C 180,E1 -4172.1,E2 -4172.1} C_VEL
LIN {X 0,Y 530.993,Z 518.341,A -85,B 0,C 180,E1 -4174.854,E2 -4174.854} C_VEL
